// TIA Portal project "Moisture_meter" (V16)

(* hardware
DEVICE "S7-1200 station_1"  S7-1200 Station
   slot 0: "Rack_0"  S7-1200 Rack  Rack  V1.0
   slot 1: "PLC_1"  CPU 1215C DC/DC/DC  6ES7 215-1AG40-0XB0  V4.4
*)

// ===== PLC "PLC_1"  CPU 1215C DC/DC/DC =====

VAR_GLOBAL   // PLC tag table "Default tag table"
   "SW1Up" AT %I0.0 : Bool;   // Концевик-1 (верх)
   "SW2Up" AT %I0.1 : Bool;   // Концевик-2 (верх)
   "SW1Down" AT %I0.2 : Bool;   // Концевик-1 (Низ)
   "SW2Down" AT %I0.3 : Bool;   // Концевик-2 (Низ)
   "modeUp" AT %I0.4 : Bool;   // Режим (верх). Авто - True
   "modeDown" AT %I0.5 : Bool;   // Режим (Низ). Авто - True
   "EmergStop" AT %I0.6 : Bool;   // Аварийный стоп
   "readyDriveUp" AT %I0.7 : Bool;   // верхний драйвер ШД - Готов
   "alarmDriveUp" AT %I1.0 : Bool;   // верхний драйвер ШД - Авария
   "readyDriveDown" AT %I1.1 : Bool;   // Нижний драйвер ШД - Готов
   "alarmDriveDown" AT %I1.2 : Bool;   // Нижний драйвер ШД - Авария
   "Axis_1_Pulse" AT %Q0.0 : Bool;   // Импульсный выход для верхнего ШД
   "Axis_1_Direction" AT %Q0.1 : Bool;   // Направление вращения для верхнего ШД
   "Axis_2_Direction" AT %Q0.4 : Bool;   // Направление вращения для Нижнего ШД
   "Axis_2_Pulse" AT %Q0.3 : Bool;   // Импульсный выход для Нижнего ШД
   "disDriveUp" AT %Q0.2 : Bool;   // дективация драйвера шагового двигателя (верх)
   "disDriveDown" AT %Q0.5 : Bool;   // дективация драйвера шагового двигателя (Низ)
   "enAir" AT %Q0.6 : Bool;   // Подача воздуха
   "Tag_1" AT %M0.0 : Bool;
   "Tag_2" AT %M0.1 : Bool;
   "Tag_3" AT %M0.2 : Bool;
   "Tag_4" AT %M0.3 : Bool;
   "Tag_5" AT %M1.0 : Bool;
   "Tag_6" AT %M1.1 : Bool;
   "Tag_7" AT %M1.2 : Bool;
   "Axis_1_DriveEnable" AT %M6.0 : Bool;   // Активация верхнего драйвера ШД
   "Axis_2_DriveEnable" AT %M6.1 : Bool;   // Активация Нижнего драйвера ШД
   "Clock_Byte" AT %MB0 : Byte;
   "Clock_10Hz" AT %M0.0 : Bool;
   "Clock_5Hz" AT %M0.1 : Bool;
   "Clock_2.5Hz" AT %M0.2 : Bool;
   "Clock_2Hz" AT %M0.3 : Bool;
   "Clock_1.25Hz" AT %M0.4 : Bool;
   "Clock_1Hz" AT %M0.5 : Bool;
   "Clock_0.625Hz" AT %M0.6 : Bool;
   "Clock_0.5Hz" AT %M0.7 : Bool;
   "System_Byte" AT %MB1 : Byte;
   "FirstScan" AT %M1.0 : Bool;
   "DiagStatusUpdate" AT %M1.1 : Bool;
   "AlwaysTRUE" AT %M1.2 : Bool;
   "AlwaysFALSE" AT %M1.3 : Bool;
   "System_Byte(1)" AT %MB1 : Byte;
   "emergStopOut" AT %M7.0 : Bool;   // Сигнал Аварийный стоп без обработки
   "emergStopDelay" AT %M7.1 : Bool;   // Сигнал Аварийный стоп, задержка после снятия
   "emergStopPRG" AT %M7.2 : Bool;   // Сигнал Аварийный стоп для останова программных блоков
   "Tag_8" AT %M10.0 : Bool;
   "Tag_9" AT %M11.0 : Bool;
   "Tag_10" AT %M11.1 : Bool;
   "Tag_11" AT %M11.2 : Bool;
   "Tag_12" AT %M11.3 : Bool;
END_VAR

DATA_BLOCK "WRITE"   // DB5
{ S7_Optimized_Access := 'FALSE' }
VERSION : 0.1
   VAR
      airBlower : Bool := false;   // обдув кожуха и обектива
      upper : Struct
         jogForward : Bool := false;   // ручное движение вперед
         jogBackward : Bool := false;   // ручное движение назад
         width : DInt := 2050;   // ширина сканирования (100~2400mm)
         delay : DInt := 100;   // Задержка перед сменой направления
         speed : DInt := 50;   // Скорость движения (1~100%)
         speedJog : DInt := 50;   // Скорость движ. в ручном режиме
         speedInitia : DInt := 50;   // Скорость инициализации
         pulsesPerMeter : DInt := 170778;   // Импульсов на 1 метр
         offsetCenter : DInt := 0;   // смещение зоны сканирования относительно центра
      END_STRUCT;
      lower : Struct
         jogForward : Bool := false;   // ручное движение вперед
         jogBackward : Bool := false;   // ручное движение назад
         width : DInt := 2050;   // ширина сканирования (100~2400mm)
         delay : DInt := 100;   // Задержка перед сменой направления
         speed : DInt := 50;   // Скорость движения (1~100%)
         speedJog : DInt := 50;   // Скорость движ. в ручном режиме
         speedInitia : DInt := 50;   // Скорость инициализации
         pulsesPerMeter : DInt := 170778;   // Импульсов на 1 метр
         offsetCenter : DInt := 0;   // смещение зоны сканирования относительно центра
      END_STRUCT;
   END_VAR
BEGIN
END_DATA_BLOCK

DATA_BLOCK "Write_buffer"   // DB10
{ S7_Optimized_Access := 'FALSE' }
VERSION : 0.1
   VAR
      airBlower : Bool := false;   // обдув кожуха и обектива
      upper : Struct
         jogForward : Bool := false;   // ручное движение вперед
         jogBackward : Bool := false;   // ручное движение назад
         width : DInt := 2050;   // ширина сканирования (100~2400mm)
         delay : DInt := 100;   // Задержка перед сменой направления
         speed : DInt := 50;   // Скорость движения (1~100%)
         speedJog : DInt := 10;   // Скорость движ. в ручном режиме
         speedInitia : DInt := 5;   // Скорость инициализации
         pulsesPerMeter : DInt := 170778;   // Импульсов на 1 метр
         offsetCenter : DInt := 0;   // смещение зоны сканирования относительно центра
      END_STRUCT;
      lower : Struct
         jogForward : Bool := false;   // ручное движение вперед
         jogBackward : Bool := false;   // ручное движение назад
         width : DInt := 2050;   // ширина сканирования (100~2400mm)
         delay : DInt := 100;   // Задержка перед сменой направления
         speed : DInt := 50;   // Скорость движения (1~100%)
         speedJog : DInt := 10;   // Скорость движ. в ручном режиме
         speedInitia : DInt := 5;   // Скорость инициализации
         pulsesPerMeter : DInt := 170778;   // Импульсов на 1 метр
         offsetCenter : DInt := 0;   // смещение зоны сканирования относительно центра
      END_STRUCT;
   END_VAR
BEGIN
END_DATA_BLOCK

DATA_BLOCK "Edit_Input"   // DB11
{ S7_Optimized_Access := 'TRUE' }
VERSION : 0.1
   VAR
      SW1UpperEdit : USInt;   // 0 - выкл, 1 - False, 2 - True Концевик верх - 1
      SW2UpperEdit : USInt := 0;   // 0 - выкл, 1 - False, 2 - True Концевик верх - 2
      SW1lowerEdit : USInt := 0;   // 0 - выкл, 1 - False, 2 - True Концевик низ - 1
      SW2lowerEdit : USInt := 0;   // 0 - выкл, 1 - False, 2 - True Концевик низ - 2
      autoUpperEdit : USInt := 0;   // 0 - выкл, 1 - False, 2 - True Режим авто верх (вкл)
      autoLowerEdit : USInt := 0;   // 0 - выкл, 1 - False, 2 - True Режим авто Низ (вкл)
      emergencyStopEdit : USInt := 0;   // 0 - выкл, 1 - False, 2 - True Аварийный стоп
      readyUpperEdit : USInt := 0;   // 0 - выкл, 1 - False, 2 - True Привод верх - готов
      alarmUpperEdit : USInt := 0;   // 0 - выкл, 1 - False, 2 - True Привод верх - авария
      readyLowerEdit : USInt := 0;   // 0 - выкл, 1 - False, 2 - True Привод Низ - готов
      alarmlowerEdit : USInt := 0;   // 0 - выкл, 1 - False, 2 - True Привод Низ - авария
   END_VAR
BEGIN
END_DATA_BLOCK

DATA_BLOCK "READ"   // DB13
{ S7_Optimized_Access := 'FALSE' }
VERSION : 0.1
   VAR
      upper : Struct
         autoEn : Bool;   // задано авто перемещение
         status : USInt;   // 0: ожидание, 1: инициализация, 2: работа, 2:авария
         distanceL1 : DInt := 0;   // расстояние от нулевой позиции до начала обЪекта измерения, мм
         distanceL2 : DInt := 0;   // ширина обЪекта измерения, мм
         speed : DInt;   // скорость перемещения верхнего, %
         currDistance : DInt;   // положение влагомера на обЪекте измерения, мм
         currMoisture : Real;   // Текущая влажность
         arrayMoisture : Array[0..99] of Real;   // Массив влажности
      END_STRUCT;
      lower : Struct
         autoEn : Bool;   // задано авто перемещение
         status : USInt;   // 0: ожидание, 1: инициализация, 2: работа, 2:авария
         distanceL1 : DInt := 0;   // расстояние от нулевой позиции до начала обЪекта измерения, мм
         distanceL2 : DInt := 0;   // ширина обЪекта измерения, мм
         speed : DInt;   // скорость перемещения верхнего, %
         currDistance : DInt;   // положение влагомера на обЪекте измерения, мм
         currMoisture : Real;   // Текущая влажность
         arrayMoisture : Array[0..99] of Real;   // Массив влажности
      END_STRUCT;
      copyDbWrite : Struct
         airBlower : Bool := false;   // обдув кожуха и обектива
         upper : Struct
            jogForward : Bool := false;   // Премещение вперед (верх влагомер)
            jogBackward : Bool := false;   // Премещение Назад (верх влагомер)
            width : DInt := 2050;   // Длина пути рабоч. зоны (верхнего)
            delay : DInt := 100;   // Задержка перед сменой направления (верх)
            speed : DInt := 50;   // Скорость верхенего (%) от HMI
            speedJog : DInt := 10;   // Скорость движ. в ручном режиме верх
            speedInitia : DInt := 5;   // Скорость движ. при инициализации верх
            pulsesPerMeter : DInt := 170778;   // Импульсов на 1 метр от HMI (верхнего)
            offsetCenter : DInt := 0;   // коррекция длины L1 (верх)
         END_STRUCT;
         lower : Struct
            jogForward : Bool := false;   // Премещение вперед (низ влагомер)
            jogBackward : Bool := false;   // Премещение Назад (низ влагомер)
            width : DInt := 2050;   // Длина пути рабоч. зоны (нижнего)
            delay : DInt := 100;   // Задержка перед сменой направления (низ)
            speed : DInt := 50;   // Скорость нижнего (%) от HMI
            speedJog : DInt := 10;   // Скорость движ. в ручном режиме низ
            speedInitia : DInt := 5;   // Скорость движ. при инициализации низ
            pulsesPerMeter : DInt := 170778;   // Импульсов на 1 метр от HMI (нижнего)
            offsetCenter : DInt := 0;   // коррекция длины L1 (низ)
         END_STRUCT;
      END_STRUCT;
   END_VAR
BEGIN
END_DATA_BLOCK

DATA_BLOCK "main_DB"   // DB63
{ S7_Optimized_Access := 'FALSE' }
VERSION : 0.1
   VAR
      SW1Up : Bool;   // Концевик верх - 1
      SW2Up : Bool;   // Концевик верх - 2
      SW1Down : Bool;   // Концевик низ - 1
      SW2Down : Bool;   // Концевик низ - 2
      autoUp : Bool;   // Режим авто активен (верх). Активация авто перемещения.
      autoDown : Bool;   // Режим авто активен (Низ). Активация авто перемещения.
      readyDriveUp : Bool;   // Привод верх - готов
      alarmDriveUp : Bool;   // Привод верх - авария
      readyDriveDown : Bool;   // Привод Низ - готов
      alarmDriveDown : Bool;   // Привод Низ - авария
      modeInitiaUp : Bool;   // Статус - идет инициализация (верх)
      modeInitiaDown : Bool;   // Статус - идет инициализация (Низ)
      modeRunUp : Bool;   // Статус - активно авто перемещение (верх)
      modeRunDown : Bool;   // Статус - активно авто перемещение (Низ)
      directionUp : Bool;   // Направление движения. True - обратно (верх)
      directionDown : Bool;   // Направление движения. True - обратно (Низ)
      initializingUp : Bool;   // Флаг - инициализация (верх)
      initializingDown : Bool;   // Флаг - инициализация (Низ)
      initialOKUP : Bool;   // Инициализация завершена (без задержки) верх
      initialOKDown : Bool;   // Инициализация завершена (без задержки) Низ
      initialOKdelayUp : Bool;   // Инициализация завершена (с запазданием) верх
      initialOKdelayDown : Bool;   // Инициализация завершена (с запазданием) Низ
      "^ChangeL1Up" : Bool;   // Импульс если изменилось число L1 (верх)
      "^ChangeL2Up" : Bool;   // Импульс если изменилось число L2 (верх)
      "^ChangeL1Down" : Bool;   // Импульс если изменилось число L1 (Низ)
      "^ChangeL2Down" : Bool;   // Импульс если изменилось число L2 (Низ)
      disConnMoistUp : Bool;
      disConnMoistDown : Bool;
      modes : USInt;   // Код режимов для верха и низа (авто/руч)
      allStatus : USInt;   // Код общего состояния программы. 1 - экстренный стоп
      statusUpHMI : USInt;   // Код состояния программы верх 0 - ожидание, 1- сработал концевик, 2 - инициализация, 3 - работа, 4 - авария привода
      statusDownHMI : USInt;   // Код состояния программы Низ 0 - ожидание, 1- сработал концевик, 2 - инициализация, 3 - работа, 4 - авария привода
      speedJogMoveUp : DInt;   // Скорость (имп/сек). Принимает значение скорости при инициализации или ручного режима
      speedJogMoveDown : DInt;   // Скорость (имп/сек). Принимает значение скорости при инициализации или ручного режима
      pulsesPerMMUp : DInt;   // Вычисленное кол-во импульсов на 1мм пути (верх)
      pulsesPerMMDown : DInt;   // Вычисленное кол-во импульсов на 1мм пути (Низ)
      setPulsesUp : DInt;   // Текущая уставка длины L (верх)
      setPulsesDown : DInt;   // Текущая уставка длины L (Низ)
      actualPulsesUp : DInt;   // Текущая уставка длины L с инверсией знака для обратного движения (верх)
      actualPulsesDown : DInt;   // Текущая уставка длины L с инверсией знака для обратного движения (НИз)
      speedPulsesUp : DInt;   // Скорость перемещения в режиме авто (имп/сек) верх
      speedPulsesDown : DInt;   // Скорость перемещения в режиме авто (имп/сек) Низ
      speedPulsesIniUp : DInt;   // Скорость перемещения при инициализации (имп/сек) верх
      speedPulsesIniDown : DInt;   // Скорость перемещения при инициализации (имп/сек) Низ
      speedPulsesJogUp : DInt;   // Скорость перемещения в ручном режиме (имп/сек) верх
      speedPulsesJogDown : DInt;   // Скорость перемещения в ручном режиме (имп/сек) Низ
   END_VAR
BEGIN
END_DATA_BLOCK

// folder: FB_blocks

DATA_BLOCK "MBTCP2_DB"   // DB2
{ S7_Optimized_Access := 'TRUE' }
VERSION : 0.1
// stored: InstanceOfName MBTCP2
"MBTCP2"
BEGIN
END_DATA_BLOCK

DATA_BLOCK "MBTCP_1_DB"   // DB3
{ S7_Optimized_Access := 'TRUE' }
VERSION : 0.1
// stored: InstanceOfName MBTCP_1
"MBTCP_1"
BEGIN
END_DATA_BLOCK

DATA_BLOCK "Moisture_up_DB"   // DB7
{ S7_Optimized_Access := 'TRUE' }
VERSION : 0.1
// stored: InstanceOfName Moisture_array
"Moisture_array"
BEGIN
END_DATA_BLOCK

DATA_BLOCK "Moisture_down_DB"   // DB8
{ S7_Optimized_Access := 'TRUE' }
VERSION : 0.1
// stored: InstanceOfName Moisture_array
"Moisture_array"
BEGIN
END_DATA_BLOCK

// folder: Socket_Send

DATA_BLOCK "Send_Connect"   // DB17
{ S7_Optimized_Access := 'TRUE' }
AUTHOR : SIMATIC
FAMILY : MC7Plus
NAME : TC_IP_v4
VERSION : 1.0
// stored: InstanceOfName TCON_IP_v4
"TCON_IP_v4"
BEGIN
   ID := 4;
   InterfaceId := 64;
   LocalPort := 2000;
END_DATA_BLOCK

DATA_BLOCK "Sock_RD_DB"   // DB19
{ S7_Optimized_Access := 'TRUE' }
VERSION : 0.1
// stored: InstanceOfName Sock_RD
"Sock_RD"
BEGIN
END_DATA_BLOCK

// folder: Socket_Write

DATA_BLOCK "Sock_WR_db"   // DB9
{ S7_Optimized_Access := 'TRUE' }
VERSION : 0.1
// stored: InstanceOfName Sock_WR
"Sock_WR"
BEGIN
END_DATA_BLOCK

DATA_BLOCK "WriteBuffer"   // DB16
{ S7_Optimized_Access := 'FALSE' }
VERSION : 0.1
   VAR
      resetErrorTrigg : Bool;   // Сброс аварии
      coolAirEn : Bool;
      setLasersManual : Struct   // Для ручного режима
         upBlueLasers123 : Bool := false;
         upGreenLasers123 : Bool := false;
         upBlueLasers456 : Bool := false;
         upGreenLasers456 : Bool := false;
         upBlueLasers789 : Bool := false;
         downGreenLasers123 : Bool := false;
         downBlueLasers123 : Bool := false;
         downGreenLasers465 : Bool := false;
         downBlueLasers456 : Bool := false;
         downGreenLasers789 : Bool := false;
      END_STRUCT;
      simulate : Struct   // Симуляция каналов. (для АО применимо из setPowerLasers)
         DI : Struct
            DI0 : USInt := 16#0;
            DI1 : USInt := 16#0;
            DI2 : USInt := 16#0;
            DI3 : USInt := 16#0;
            DI4 : USInt := 16#0;
            DI5 : USInt := 16#0;
            DI6 : USInt := 16#0;
            DI7 : USInt := 16#0;
            DI8 : USInt := 16#0;
            DI9 : USInt := 16#0;
            DI10 : USInt := 16#0;
            DI11 : USInt := 16#0;
            DI12 : USInt := 16#0;
            DI13 : USInt := 16#0;
            DI14 : USInt := 16#0;
            DI15 : USInt := 16#0;
         END_STRUCT;
         "DO" : Struct
            DO0 : USInt := 0;
            DO1 : USInt := 0;
            DO2 : USInt := 0;
            DO3 : USInt := 0;
            DO4 : USInt := 0;
            DO5 : USInt := 0;
            DO6 : USInt := 0;
            DO7 : USInt := 0;
            DO8 : USInt := 0;
            DO9 : USInt := 0;
            DO10 : USInt := 0;
            DO11 : USInt := 0;
            DO12 : USInt := 0;
            DO13 : USInt := 0;
            DO14 : USInt := 0;
            DO15 : USInt := 0;
            DO16 : USInt := 0;
            DO17 : USInt := 0;
            DO18 : USInt := 0;
            DO19 : USInt := 0;
            DO20 : USInt := 0;
            DO21 : USInt := 0;
            DO22 : USInt := 0;
            DO23 : USInt := 0;
            DO24 : USInt := 0;
            DO25 : USInt := 0;
            DO26 : USInt := 0;
            DO27 : USInt := 0;
            DO28 : USInt := 0;
            DO29 : USInt := 0;
            DO30 : USInt := 0;
            DO31 : USInt := 0;
         END_STRUCT;
         AI : Struct   // 0.0 -- симуляция отключена; от 0.0 до 0.001 -- запись 0.0; выше 0.001 -- запись любого числа.
            upTempLaser1 : Real := 0.0;
            upTempLaser2 : Real := 0.0;
            upTempCam1 : Real := 0.0;
            upTempCam2 : Real := 0.0;
            downTempLaser1 : Real := 0.0;
            downTempLaser2 : Real := 0.0;
            downTempCam1 : Real := 0.0;
            downTempCam2 : Real := 0.0;
            airTemperatur : Real := 0.0;
            reserv : Real := 0.0;
         END_STRUCT;
      END_STRUCT;
      setTemperatures : Struct   // Уставки температур
         faultUpLaser : Real := 0.0;
         faultUpCam : Real := 0.0;
         faultDownLaser : Real := 0.0;
         faultDownCam : Real := 0.0;
         warnAir : Real := 0.0;
         warnUpLaser : Real := 0.0;
         warnUpCam : Real := 0.0;
         warnDownLaser : Real := 0.0;
         warnDownCam : Real := 0.0;
         reserv0 : Real := 0.0;
      END_STRUCT;
      cleanTime : Struct   // Периодичность продувки
         tOnS : Real := 0.0;
         tOffMin : Real := 0.0;
      END_STRUCT;
      setPowerLasers : Struct   // Мощность лазеров (0 -- 100%)
         writeAll : Real := 0.0;
         upBlue1 : Real := 0.0;   // AO0.0
         upBlue2 : Real := 0.0;   // AO0.1
         upBlue3 : Real := 0.0;   // AO0.2
         upGreen1 : Real := 0.0;   // AO0.3
         upGreen2 : Real := 0.0;   // AO0.4
         upGreen3 : Real := 0.0;   // AO0.5
         upBlue4 : Real := 0.0;   // AO0.6
         upBlue5 : Real := 0.0;   // AO0.7
         upBlue6 : Real := 0.0;   // AO1.0
         upGreen4 : Real := 0.0;   // AO1.1
         upGreen5 : Real := 0.0;   // AO1.2
         upGreen6 : Real := 0.0;   // AO1.3
         upBlue7 : Real := 0.0;   // AO1.4
         upBlue8 : Real := 0.0;   // AO1.5
         upBlue9 : Real := 0.0;   // AO1.6
         downGreen1 : Real := 0.0;   // AO2.0
         downGreen2 : Real := 0.0;   // AO2.1
         downGreen3 : Real := 0.0;   // AO2.2
         downBlue1 : Real := 0.0;   // AO2.3
         downBlue2 : Real := 0.0;   // AO2.4
         downBlue3 : Real := 0.0;   // AO2.5
         downGreen4 : Real := 0.0;   // AO2.6
         downGreen5 : Real := 0.0;   // AO2.7
         downGreen6 : Real := 0.0;   // AO3.0
         downBlue4 : Real := 0.0;   // AO3.1
         downBlue5 : Real := 0.0;   // AO3.2
         downBlue6 : Real := 0.0;   // AO3.3
         downGreen7 : Real := 0.0;   // AO3.4
         downGreen8 : Real := 0.0;   // AO3.5
         downGreen9 : Real := 0.0;   // AO3.6
      END_STRUCT;
   END_VAR
BEGIN
END_DATA_BLOCK

DATA_BLOCK "TRCV_Connect"   // DB20
{ S7_Optimized_Access := 'TRUE' }
AUTHOR : SIMATIC
FAMILY : MC7Plus
NAME : TC_IP_v4
VERSION : 1.0
// stored: InstanceOfName TCON_IP_v4
"TCON_IP_v4"
BEGIN
   ID := 3;
   InterfaceId := 64;
   LocalPort := 2001;
END_DATA_BLOCK

// folder: System blocks/Program resources

DATA_BLOCK "IEC_Timer_0_DB"   // DB14
{ S7_Optimized_Access := 'TRUE' }
AUTHOR : Simatic
FAMILY : IEC
NAME : IEC_TMR
VERSION : 1.0
// stored: InstanceOfName IEC_TIMER
"IEC_TIMER"
BEGIN
END_DATA_BLOCK

DATA_BLOCK "IEC_Timer_0_DB_1"   // DB15
{ S7_Optimized_Access := 'TRUE' }
AUTHOR : Simatic
FAMILY : IEC
NAME : IEC_TMR
VERSION : 1.0
// stored: InstanceOfName IEC_TIMER
"IEC_TIMER"
BEGIN
END_DATA_BLOCK

// folder: initializing

DATA_BLOCK "initializingUP_DB"   // DB12
{ S7_Optimized_Access := 'TRUE' }
VERSION : 0.1
// stored: InstanceOfName initializing
"initializing"
BEGIN
END_DATA_BLOCK

DATA_BLOCK "initializingDown_DB"   // DB60
{ S7_Optimized_Access := 'TRUE' }
VERSION : 0.1
// stored: InstanceOfName initializing
"initializing"
BEGIN
END_DATA_BLOCK

// folder: math

DATA_BLOCK "math_DB"   // DB25
{ S7_Optimized_Access := 'TRUE' }
VERSION : 0.1
// stored: InstanceOfName math
"math"
BEGIN
END_DATA_BLOCK

// folder: moving

DATA_BLOCK "movingUp_DB"   // DB26
{ S7_Optimized_Access := 'TRUE' }
VERSION : 0.1
// stored: InstanceOfName moving
"moving"
BEGIN
END_DATA_BLOCK

DATA_BLOCK "movingDown_DB"   // DB27
{ S7_Optimized_Access := 'TRUE' }
VERSION : 0.1
// stored: InstanceOfName moving
"moving"
BEGIN
END_DATA_BLOCK

// folder: status&Mode

DATA_BLOCK "statusMove_DB"   // DB4
{ S7_Optimized_Access := 'TRUE' }
VERSION : 0.1
// stored: InstanceOfName statusMove
"statusMove"
BEGIN
END_DATA_BLOCK

// folder: (top level)

DATA_BLOCK "AxisUpper"   // DB1, Motion_DB
{ S7_Optimized_Access := 'TRUE' }
AUTHOR : SIMATIC
FAMILY : BasicMC
NAME : TO_PosAx
VERSION : 7.0
// stored: InstanceOfName TO_PositioningAxis
"TO_PositioningAxis"
BEGIN
   // Axis.EnableOutput_AddressCU = %M6.0
   // Axis.DirectionOutputEnabledCU = TRUE
   // Axis.OnlinePtoModeCU = 16#0000_0002
   // Axis.SelectedChannel2EnumCU = %Q0.1
   // Axis.SelectedChannel1EnumCU = %Q0.0
   // Pulse.MinDeltaDeltaFrequencyCU = 0.004
   // Pulse.MaxDeltaDeltaFrequencyCU = 1.0E+10
   // Pulse.MinDeltaFrequencyCU = 0.005
   // Pulse.MaxDeltaFrequencyCU = 9.5E+9
   // Pulse.MinFrequencyCU = 1.0
   // Pulse.MaxFrequencyCU = 100000.0
   // Pulse.OutputSourceCU = 16#0000_0000
   // Axis.SelectPTO = 0
   // Axis.LengthUnit.LastDistance = -1
END_DATA_BLOCK

DATA_BLOCK "AxisLower"   // DB6, Motion_DB
{ S7_Optimized_Access := 'TRUE' }
AUTHOR : SIMATIC
FAMILY : BasicMC
NAME : TO_PosAx
VERSION : 7.0
// stored: InstanceOfName TO_PositioningAxis
"TO_PositioningAxis"
BEGIN
   // Axis.EnableOutput_AddressCU = %M6.1
   // Axis.LengthUnit.LastDistance = -1
   // Axis.DirectionOutputEnabledCU = TRUE
   // Axis.OnlinePtoModeCU = 16#0000_0002
   // Axis.SelectedChannel2EnumCU = %Q0.4
   // Axis.SelectedChannel1EnumCU = %Q0.3
   // Pulse.MinDeltaDeltaFrequencyCU = 0.004
   // Pulse.MaxDeltaDeltaFrequencyCU = 1.0E+10
   // Pulse.MinDeltaFrequencyCU = 0.005
   // Pulse.MaxDeltaFrequencyCU = 9.5E+9
   // Pulse.MinFrequencyCU = 1.0
   // Pulse.MaxFrequencyCU = 100000.0
   // Pulse.OutputSourceCU = 16#0000_0000
   // Axis.SelectPTO = 1
   // Axis.OnlinePtoIndexCU = 1
END_DATA_BLOCK

ORGANIZATION_BLOCK "Main"   // OB1, LAD, ProgramCycle
{ S7_Optimized_Access := 'TRUE' }
VERSION : 0.1
   VAR_INPUT
      Initial_Call : Bool;   // Initial call of this OB
      Remanence : Bool;   // =True, if remanent data are available
   END_VAR
BEGIN

REGION Network 1: Ручное изменение состояния дискретных входов контроллера
   // Значения хранятся в блоке Edit_Input [DB11]:    0 - выкл, 1 - False, 2 - True
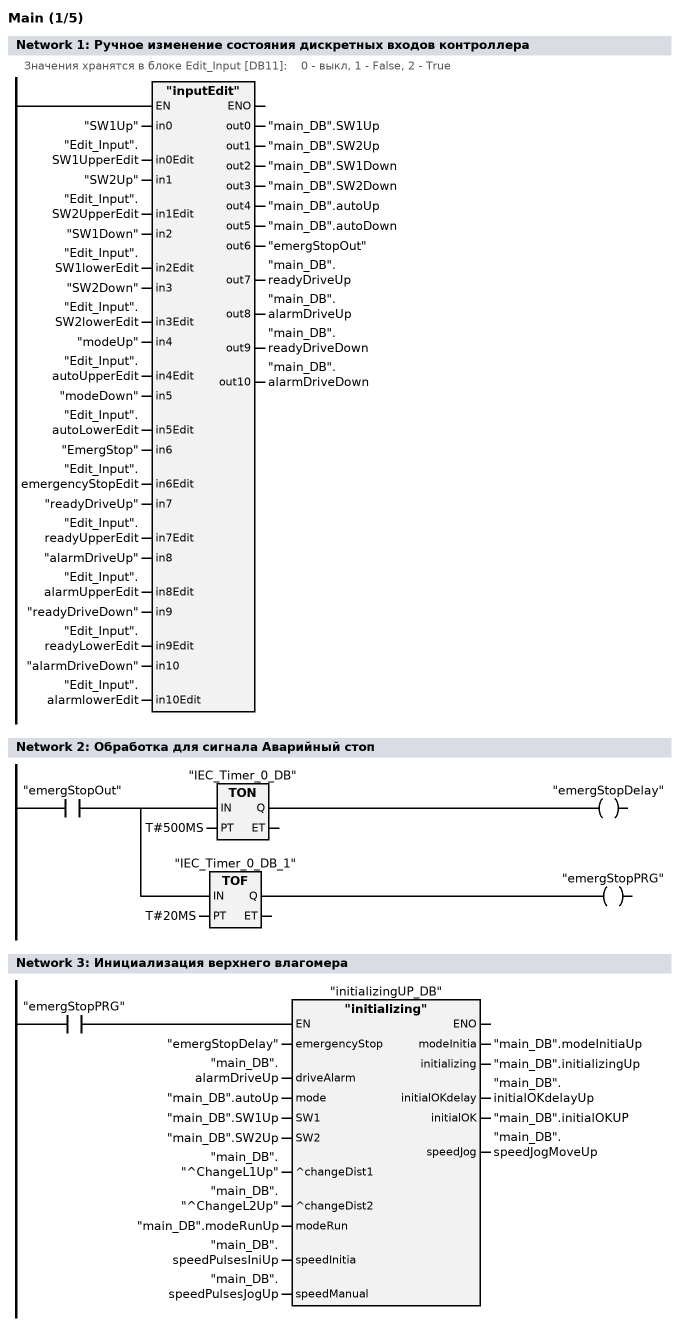
   RUNG wire#powerrail
      "inputEdit"(in0 := "SW1Up", in0Edit := "Edit_Input".SW1UpperEdit, in1 := "SW2Up", in1Edit := "Edit_Input".SW2UpperEdit, in2 := "SW1Down", in2Edit := "Edit_Input".SW1lowerEdit, in3 := "SW2Down", in3Edit := "Edit_Input".SW2lowerEdit, in4 := "modeUp", in4Edit := "Edit_Input".autoUpperEdit, in5 := "modeDown", in5Edit := "Edit_Input".autoLowerEdit, in6 := "EmergStop", in6Edit := "Edit_Input".emergencyStopEdit, in7 := "readyDriveUp", in7Edit := "Edit_Input".readyUpperEdit, in8 := "alarmDriveUp", in8Edit := "Edit_Input".alarmUpperEdit, in9 := "readyDriveDown", in9Edit := "Edit_Input".readyLowerEdit, in10 := "alarmDriveDown", in10Edit := "Edit_Input".alarmlowerEdit, out0 => "main_DB".SW1Up, out1 => "main_DB".SW2Up, out2 => "main_DB".SW1Down, out3 => "main_DB".SW2Down, out4 => "main_DB".autoUp, out5 => "main_DB".autoDown, out6 => "emergStopOut", out7 => "main_DB".readyDriveUp, out8 => "main_DB".alarmDriveUp, out9 => "main_DB".readyDriveDown, out10 => "main_DB".alarmDriveDown)
   END_RUNG
   // the same network as SCL:
   "inputEdit"(in0 := "SW1Up",
               in0Edit := "Edit_Input".SW1UpperEdit,
               in1 := "SW2Up",
               in1Edit := "Edit_Input".SW2UpperEdit,
               in2 := "SW1Down",
               in2Edit := "Edit_Input".SW1lowerEdit,
               in3 := "SW2Down",
               in3Edit := "Edit_Input".SW2lowerEdit,
               in4 := "modeUp",
               in4Edit := "Edit_Input".autoUpperEdit,
               in5 := "modeDown",
               in5Edit := "Edit_Input".autoLowerEdit,
               in6 := "EmergStop",
               in6Edit := "Edit_Input".emergencyStopEdit,
               in7 := "readyDriveUp",
               in7Edit := "Edit_Input".readyUpperEdit,
               in8 := "alarmDriveUp",
               in8Edit := "Edit_Input".alarmUpperEdit,
               in9 := "readyDriveDown",
               in9Edit := "Edit_Input".readyLowerEdit,
               in10 := "alarmDriveDown",
               in10Edit := "Edit_Input".alarmlowerEdit,
               out0 => "main_DB".SW1Up,
               out1 => "main_DB".SW2Up,
               out2 => "main_DB".SW1Down,
               out3 => "main_DB".SW2Down,
               out4 => "main_DB".autoUp,
               out5 => "main_DB".autoDown,
               out6 => "emergStopOut",
               out7 => "main_DB".readyDriveUp,
               out8 => "main_DB".alarmDriveUp,
               out9 => "main_DB".readyDriveDown,
               out10 => "main_DB".alarmDriveDown);
END_REGION

REGION Network 2: Обработка для сигнала Аварийный стоп
   "IEC_Timer_0_DB".TON(IN := "emergStopOut", PT := T#500MS);
   "emergStopDelay" := "IEC_Timer_0_DB".Q;
   "IEC_Timer_0_DB_1".TOF(IN := "emergStopOut", PT := T#20MS);
   "emergStopPRG" := "IEC_Timer_0_DB_1".Q;
END_REGION

REGION Network 3: Инициализация верхнего влагомера
   RUNG wire#powerrail
      Contact( "emergStopPRG" )
      "initializingUP_DB"(emergencyStop := "emergStopDelay", driveAlarm := "main_DB".alarmDriveUp, mode := "main_DB".autoUp, SW1 := "main_DB".SW1Up, SW2 := "main_DB".SW2Up, "^changeDist1" := "main_DB"."^ChangeL1Up", "^changeDist2" := "main_DB"."^ChangeL2Up", modeRun := "main_DB".modeRunUp, speedInitia := "main_DB".speedPulsesIniUp, speedManual := "main_DB".speedPulsesJogUp, modeInitia => "main_DB".modeInitiaUp, initializing => "main_DB".initializingUp, initialOKdelay => "main_DB".initialOKdelayUp, initialOK => "main_DB".initialOKUP, speedJog => "main_DB".speedJogMoveUp)
   END_RUNG
   // the same network as SCL:
   IF "emergStopPRG" THEN
       "initializingUP_DB"(emergencyStop := "emergStopDelay",   // "initializing"
                           driveAlarm := "main_DB".alarmDriveUp,
                           mode := "main_DB".autoUp,
                           SW1 := "main_DB".SW1Up,
                           SW2 := "main_DB".SW2Up,
                           "^changeDist1" := "main_DB"."^ChangeL1Up",
                           "^changeDist2" := "main_DB"."^ChangeL2Up",
                           modeRun := "main_DB".modeRunUp,
                           speedInitia := "main_DB".speedPulsesIniUp,
                           speedManual := "main_DB".speedPulsesJogUp,
                           modeInitia => "main_DB".modeInitiaUp,
                           initializing => "main_DB".initializingUp,
                           initialOKdelay => "main_DB".initialOKdelayUp,
                           initialOK => "main_DB".initialOKUP,
                           speedJog => "main_DB".speedJogMoveUp);
   END_IF;
END_REGION

REGION Network 4: Инициализация нижнего влагомера
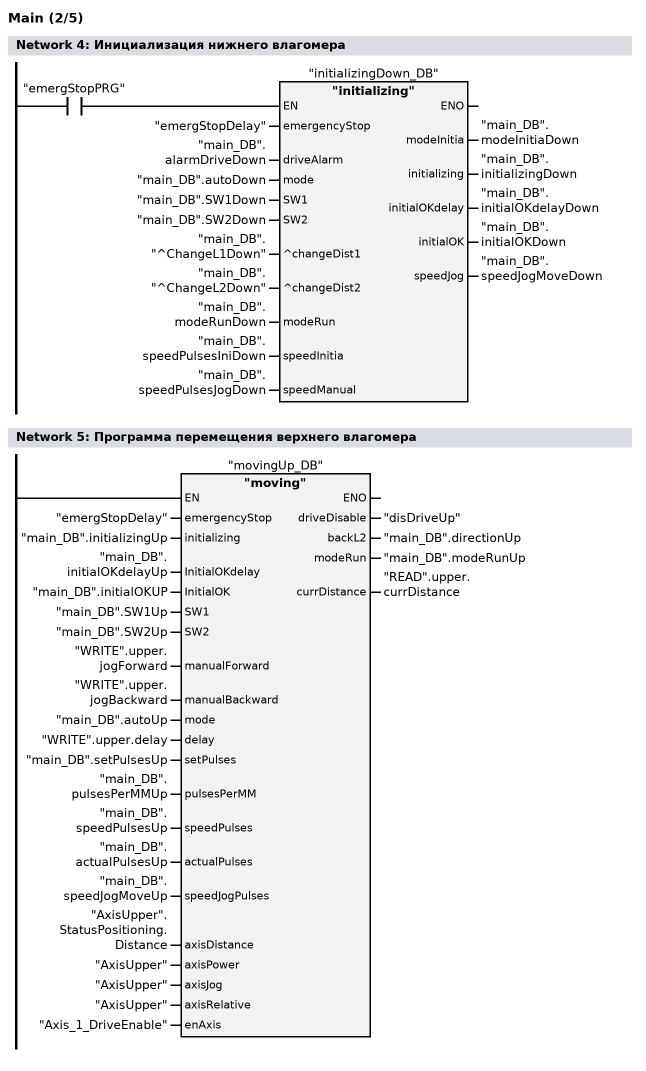
   RUNG wire#powerrail
      Contact( "emergStopPRG" )
      "initializingDown_DB"(emergencyStop := "emergStopDelay", driveAlarm := "main_DB".alarmDriveDown, mode := "main_DB".autoDown, SW1 := "main_DB".SW1Down, SW2 := "main_DB".SW2Down, "^changeDist1" := "main_DB"."^ChangeL1Down", "^changeDist2" := "main_DB"."^ChangeL2Down", modeRun := "main_DB".modeRunDown, speedInitia := "main_DB".speedPulsesIniDown, speedManual := "main_DB".speedPulsesJogDown, modeInitia => "main_DB".modeInitiaDown, initializing => "main_DB".initializingDown, initialOKdelay => "main_DB".initialOKdelayDown, initialOK => "main_DB".initialOKDown, speedJog => "main_DB".speedJogMoveDown)
   END_RUNG
   // the same network as SCL:
   IF "emergStopPRG" THEN
       "initializingDown_DB"(emergencyStop := "emergStopDelay",   // "initializing"
                             driveAlarm := "main_DB".alarmDriveDown,
                             mode := "main_DB".autoDown,
                             SW1 := "main_DB".SW1Down,
                             SW2 := "main_DB".SW2Down,
                             "^changeDist1" := "main_DB"."^ChangeL1Down",
                             "^changeDist2" := "main_DB"."^ChangeL2Down",
                             modeRun := "main_DB".modeRunDown,
                             speedInitia := "main_DB".speedPulsesIniDown,
                             speedManual := "main_DB".speedPulsesJogDown,
                             modeInitia => "main_DB".modeInitiaDown,
                             initializing => "main_DB".initializingDown,
                             initialOKdelay => "main_DB".initialOKdelayDown,
                             initialOK => "main_DB".initialOKDown,
                             speedJog => "main_DB".speedJogMoveDown);
   END_IF;
END_REGION

REGION Network 5: Программа перемещения верхнего влагомера
   RUNG wire#powerrail
      "movingUp_DB"(emergencyStop := "emergStopDelay", initializing := "main_DB".initializingUp, InitialOKdelay := "main_DB".initialOKdelayUp, InitialOK := "main_DB".initialOKUP, SW1 := "main_DB".SW1Up, SW2 := "main_DB".SW2Up, manualForward := "WRITE".upper.jogForward, manualBackward := "WRITE".upper.jogBackward, mode := "main_DB".autoUp, delay := "WRITE".upper.delay, setPulses := "main_DB".setPulsesUp, pulsesPerMM := "main_DB".pulsesPerMMUp, speedPulses := "main_DB".speedPulsesUp, actualPulses := "main_DB".actualPulsesUp, speedJogPulses := "main_DB".speedJogMoveUp, axisDistance := "AxisUpper".StatusPositioning.Distance, axisPower := "AxisUpper", axisJog := "AxisUpper", axisRelative := "AxisUpper", enAxis := "Axis_1_DriveEnable", driveDisable => "disDriveUp", backL2 => "main_DB".directionUp, modeRun => "main_DB".modeRunUp, currDistance => "READ".upper.currDistance)
   END_RUNG
   // the same network as SCL:
   "movingUp_DB"(emergencyStop := "emergStopDelay",   // "moving"
                 initializing := "main_DB".initializingUp,
                 InitialOKdelay := "main_DB".initialOKdelayUp,
                 InitialOK := "main_DB".initialOKUP,
                 SW1 := "main_DB".SW1Up,
                 SW2 := "main_DB".SW2Up,
                 manualForward := "WRITE".upper.jogForward,
                 manualBackward := "WRITE".upper.jogBackward,
                 mode := "main_DB".autoUp,
                 delay := "WRITE".upper.delay,
                 setPulses := "main_DB".setPulsesUp,
                 pulsesPerMM := "main_DB".pulsesPerMMUp,
                 speedPulses := "main_DB".speedPulsesUp,
                 actualPulses := "main_DB".actualPulsesUp,
                 speedJogPulses := "main_DB".speedJogMoveUp,
                 axisDistance := "AxisUpper".StatusPositioning.Distance,
                 axisPower := "AxisUpper",
                 axisJog := "AxisUpper",
                 axisRelative := "AxisUpper",
                 enAxis := "Axis_1_DriveEnable",
                 driveDisable => "disDriveUp",
                 backL2 => "main_DB".directionUp,
                 modeRun => "main_DB".modeRunUp,
                 currDistance => "READ".upper.currDistance);
END_REGION

REGION Network 6: Программа перемещения нижнего влагомера
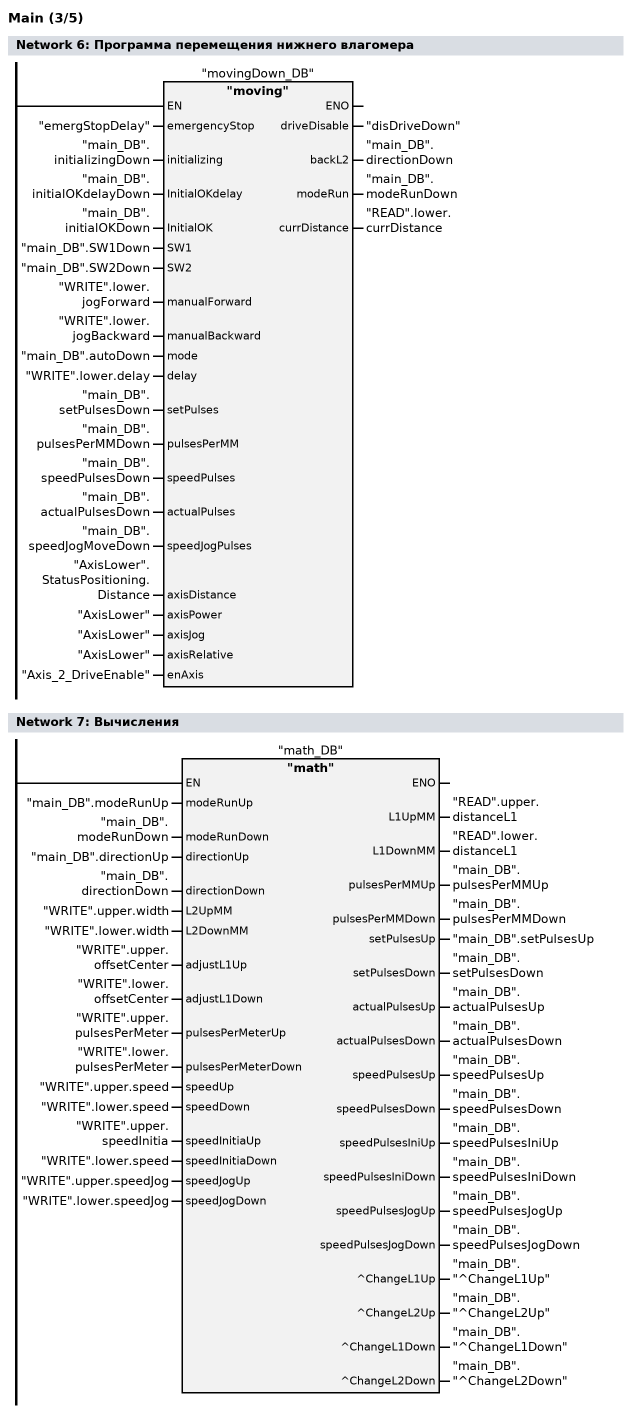
   RUNG wire#powerrail
      "movingDown_DB"(emergencyStop := "emergStopDelay", initializing := "main_DB".initializingDown, InitialOKdelay := "main_DB".initialOKdelayDown, InitialOK := "main_DB".initialOKDown, SW1 := "main_DB".SW1Down, SW2 := "main_DB".SW2Down, manualForward := "WRITE".lower.jogForward, manualBackward := "WRITE".lower.jogBackward, mode := "main_DB".autoDown, delay := "WRITE".lower.delay, setPulses := "main_DB".setPulsesDown, pulsesPerMM := "main_DB".pulsesPerMMDown, speedPulses := "main_DB".speedPulsesDown, actualPulses := "main_DB".actualPulsesDown, speedJogPulses := "main_DB".speedJogMoveDown, axisDistance := "AxisLower".StatusPositioning.Distance, axisPower := "AxisLower", axisJog := "AxisLower", axisRelative := "AxisLower", enAxis := "Axis_2_DriveEnable", driveDisable => "disDriveDown", backL2 => "main_DB".directionDown, modeRun => "main_DB".modeRunDown, currDistance => "READ".lower.currDistance)
   END_RUNG
   // the same network as SCL:
   "movingDown_DB"(emergencyStop := "emergStopDelay",   // "moving"
                   initializing := "main_DB".initializingDown,
                   InitialOKdelay := "main_DB".initialOKdelayDown,
                   InitialOK := "main_DB".initialOKDown,
                   SW1 := "main_DB".SW1Down,
                   SW2 := "main_DB".SW2Down,
                   manualForward := "WRITE".lower.jogForward,
                   manualBackward := "WRITE".lower.jogBackward,
                   mode := "main_DB".autoDown,
                   delay := "WRITE".lower.delay,
                   setPulses := "main_DB".setPulsesDown,
                   pulsesPerMM := "main_DB".pulsesPerMMDown,
                   speedPulses := "main_DB".speedPulsesDown,
                   actualPulses := "main_DB".actualPulsesDown,
                   speedJogPulses := "main_DB".speedJogMoveDown,
                   axisDistance := "AxisLower".StatusPositioning.Distance,
                   axisPower := "AxisLower",
                   axisJog := "AxisLower",
                   axisRelative := "AxisLower",
                   enAxis := "Axis_2_DriveEnable",
                   driveDisable => "disDriveDown",
                   backL2 => "main_DB".directionDown,
                   modeRun => "main_DB".modeRunDown,
                   currDistance => "READ".lower.currDistance);
END_REGION

REGION Network 7: Вычисления
   RUNG wire#powerrail
      "math_DB"(modeRunUp := "main_DB".modeRunUp, modeRunDown := "main_DB".modeRunDown, directionUp := "main_DB".directionUp, directionDown := "main_DB".directionDown, L2UpMM := "WRITE".upper.width, L2DownMM := "WRITE".lower.width, adjustL1Up := "WRITE".upper.offsetCenter, adjustL1Down := "WRITE".lower.offsetCenter, pulsesPerMeterUp := "WRITE".upper.pulsesPerMeter, pulsesPerMeterDown := "WRITE".lower.pulsesPerMeter, speedUp := "WRITE".upper.speed, speedDown := "WRITE".lower.speed, speedInitiaUp := "WRITE".upper.speedInitia, speedInitiaDown := "WRITE".lower.speed, speedJogUp := "WRITE".upper.speedJog, speedJogDown := "WRITE".lower.speedJog, L1UpMM => "READ".upper.distanceL1, L1DownMM => "READ".lower.distanceL1, pulsesPerMMUp => "main_DB".pulsesPerMMUp, pulsesPerMMDown => "main_DB".pulsesPerMMDown, setPulsesUp => "main_DB".setPulsesUp, setPulsesDown => "main_DB".setPulsesDown, actualPulsesUp => "main_DB".actualPulsesUp, actualPulsesDown => "main_DB".actualPulsesDown, speedPulsesUp => "main_DB".speedPulsesUp, speedPulsesDown => "main_DB".speedPulsesDown, speedPulsesIniUp => "main_DB".speedPulsesIniUp, speedPulsesIniDown => "main_DB".speedPulsesIniDown, speedPulsesJogUp => "main_DB".speedPulsesJogUp, speedPulsesJogDown => "main_DB".speedPulsesJogDown, "^ChangeL1Up" => "main_DB"."^ChangeL1Up", "^ChangeL2Up" => "main_DB"."^ChangeL2Up", "^ChangeL1Down" => "main_DB"."^ChangeL1Down", "^ChangeL2Down" => "main_DB"."^ChangeL2Down")
   END_RUNG
   // the same network as SCL:
   "math_DB"(modeRunUp := "main_DB".modeRunUp,   // "math"
             modeRunDown := "main_DB".modeRunDown,
             directionUp := "main_DB".directionUp,
             directionDown := "main_DB".directionDown,
             L2UpMM := "WRITE".upper.width,
             L2DownMM := "WRITE".lower.width,
             adjustL1Up := "WRITE".upper.offsetCenter,
             adjustL1Down := "WRITE".lower.offsetCenter,
             pulsesPerMeterUp := "WRITE".upper.pulsesPerMeter,
             pulsesPerMeterDown := "WRITE".lower.pulsesPerMeter,
             speedUp := "WRITE".upper.speed,
             speedDown := "WRITE".lower.speed,
             speedInitiaUp := "WRITE".upper.speedInitia,
             speedInitiaDown := "WRITE".lower.speed,
             speedJogUp := "WRITE".upper.speedJog,
             speedJogDown := "WRITE".lower.speedJog,
             L1UpMM => "READ".upper.distanceL1,
             L1DownMM => "READ".lower.distanceL1,
             pulsesPerMMUp => "main_DB".pulsesPerMMUp,
             pulsesPerMMDown => "main_DB".pulsesPerMMDown,
             setPulsesUp => "main_DB".setPulsesUp,
             setPulsesDown => "main_DB".setPulsesDown,
             actualPulsesUp => "main_DB".actualPulsesUp,
             actualPulsesDown => "main_DB".actualPulsesDown,
             speedPulsesUp => "main_DB".speedPulsesUp,
             speedPulsesDown => "main_DB".speedPulsesDown,
             speedPulsesIniUp => "main_DB".speedPulsesIniUp,
             speedPulsesIniDown => "main_DB".speedPulsesIniDown,
             speedPulsesJogUp => "main_DB".speedPulsesJogUp,
             speedPulsesJogDown => "main_DB".speedPulsesJogDown,
             "^ChangeL1Up" => "main_DB"."^ChangeL1Up",
             "^ChangeL2Up" => "main_DB"."^ChangeL2Up",
             "^ChangeL1Down" => "main_DB"."^ChangeL1Down",
             "^ChangeL2Down" => "main_DB"."^ChangeL2Down");
END_REGION

REGION Network 8: Статусы программ и передача между блоками данных
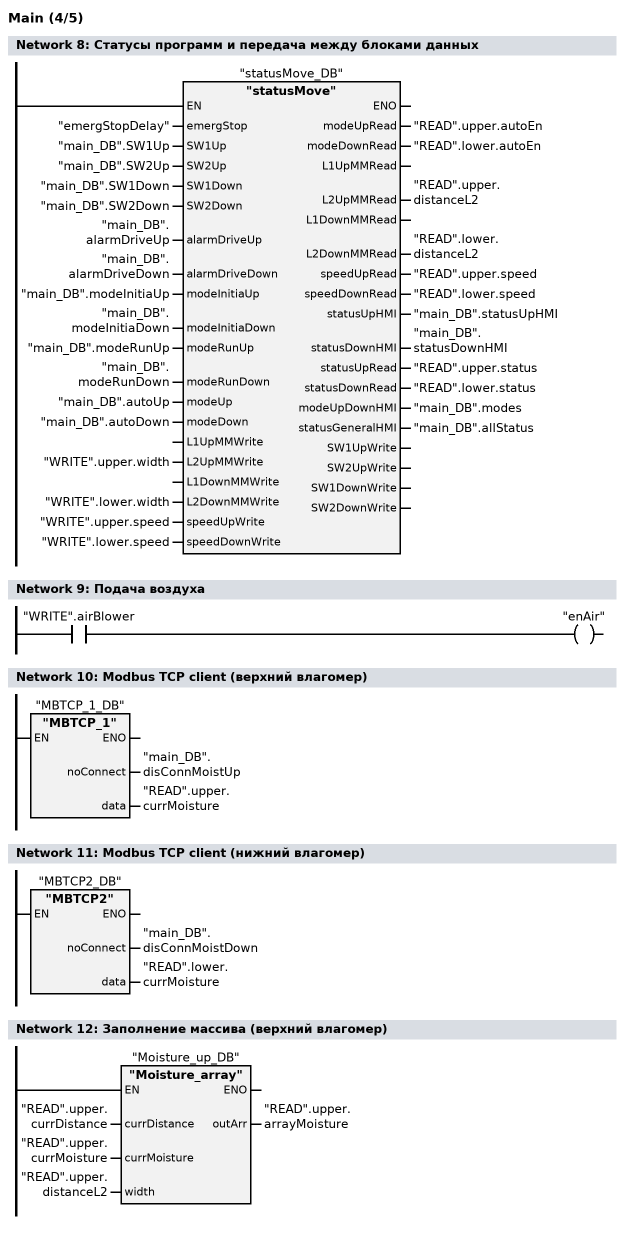
   RUNG wire#powerrail
      "statusMove_DB"(emergStop := "emergStopDelay", SW1Up := "main_DB".SW1Up, SW2Up := "main_DB".SW2Up, SW1Down := "main_DB".SW1Down, SW2Down := "main_DB".SW2Down, alarmDriveUp := "main_DB".alarmDriveUp, alarmDriveDown := "main_DB".alarmDriveDown, modeInitiaUp := "main_DB".modeInitiaUp, modeInitiaDown := "main_DB".modeInitiaDown, modeRunUp := "main_DB".modeRunUp, modeRunDown := "main_DB".modeRunDown, modeUp := "main_DB".autoUp, modeDown := "main_DB".autoDown, L1UpMMWrite :=, L2UpMMWrite := "WRITE".upper.width, L1DownMMWrite :=, L2DownMMWrite := "WRITE".lower.width, speedUpWrite := "WRITE".upper.speed, speedDownWrite := "WRITE".lower.speed, modeUpRead => "READ".upper.autoEn, modeDownRead => "READ".lower.autoEn, L1UpMMRead =>, L2UpMMRead => "READ".upper.distanceL2, L1DownMMRead =>, L2DownMMRead => "READ".lower.distanceL2, speedUpRead => "READ".upper.speed, speedDownRead => "READ".lower.speed, statusUpHMI => "main_DB".statusUpHMI, statusDownHMI => "main_DB".statusDownHMI, statusUpRead => "READ".upper.status, statusDownRead => "READ".lower.status, modeUpDownHMI => "main_DB".modes, statusGeneralHMI => "main_DB".allStatus, SW1UpWrite =>, SW2UpWrite =>, SW1DownWrite =>, SW2DownWrite =>)
   END_RUNG
   // the same network as SCL:
   "statusMove_DB"(emergStop := "emergStopDelay",   // "statusMove"
                   SW1Up := "main_DB".SW1Up,
                   SW2Up := "main_DB".SW2Up,
                   SW1Down := "main_DB".SW1Down,
                   SW2Down := "main_DB".SW2Down,
                   alarmDriveUp := "main_DB".alarmDriveUp,
                   alarmDriveDown := "main_DB".alarmDriveDown,
                   modeInitiaUp := "main_DB".modeInitiaUp,
                   modeInitiaDown := "main_DB".modeInitiaDown,
                   modeRunUp := "main_DB".modeRunUp,
                   modeRunDown := "main_DB".modeRunDown,
                   modeUp := "main_DB".autoUp,
                   modeDown := "main_DB".autoDown,
                   L2UpMMWrite := "WRITE".upper.width,
                   L2DownMMWrite := "WRITE".lower.width,
                   speedUpWrite := "WRITE".upper.speed,
                   speedDownWrite := "WRITE".lower.speed,
                   modeUpRead => "READ".upper.autoEn,
                   modeDownRead => "READ".lower.autoEn,
                   L2UpMMRead => "READ".upper.distanceL2,
                   L2DownMMRead => "READ".lower.distanceL2,
                   speedUpRead => "READ".upper.speed,
                   speedDownRead => "READ".lower.speed,
                   statusUpHMI => "main_DB".statusUpHMI,
                   statusDownHMI => "main_DB".statusDownHMI,
                   statusUpRead => "READ".upper.status,
                   statusDownRead => "READ".lower.status,
                   modeUpDownHMI => "main_DB".modes,
                   statusGeneralHMI => "main_DB".allStatus);
END_REGION

REGION Network 9: Подача воздуха
   RUNG wire#powerrail
      Contact( "WRITE".airBlower )
      Coil( "enAir" )
   END_RUNG
   // the same network as SCL:
   "enAir" := "WRITE".airBlower;
END_REGION

REGION Network 10: Modbus TCP client (верхний влагомер)
   RUNG wire#powerrail
      "MBTCP_1_DB"(noConnect => "main_DB".disConnMoistUp, data => "READ".upper.currMoisture)
   END_RUNG
   // the same network as SCL:
   "MBTCP_1_DB"(noConnect => "main_DB".disConnMoistUp, data => "READ".upper.currMoisture);   // "MBTCP_1"
END_REGION

REGION Network 11: Modbus TCP client (нижний влагомер)
   RUNG wire#powerrail
      "MBTCP2_DB"(noConnect => "main_DB".disConnMoistDown, data => "READ".lower.currMoisture)
   END_RUNG
   // the same network as SCL:
   "MBTCP2_DB"(noConnect => "main_DB".disConnMoistDown, data => "READ".lower.currMoisture);   // "MBTCP2"
END_REGION

REGION Network 12: Заполнение массива (верхний влагомер)
   RUNG wire#powerrail
      "Moisture_up_DB"(currDistance := "READ".upper.currDistance, currMoisture := "READ".upper.currMoisture, width := "READ".upper.distanceL2, outArr => "READ".upper.arrayMoisture)
   END_RUNG
   // the same network as SCL:
   "Moisture_up_DB"(currDistance := "READ".upper.currDistance,   // "Moisture_array"
                    currMoisture := "READ".upper.currMoisture,
                    width := "READ".upper.distanceL2,
                    outArr => "READ".upper.arrayMoisture);
END_REGION

REGION Network 13: Заполнение массива (нижний влагомер)
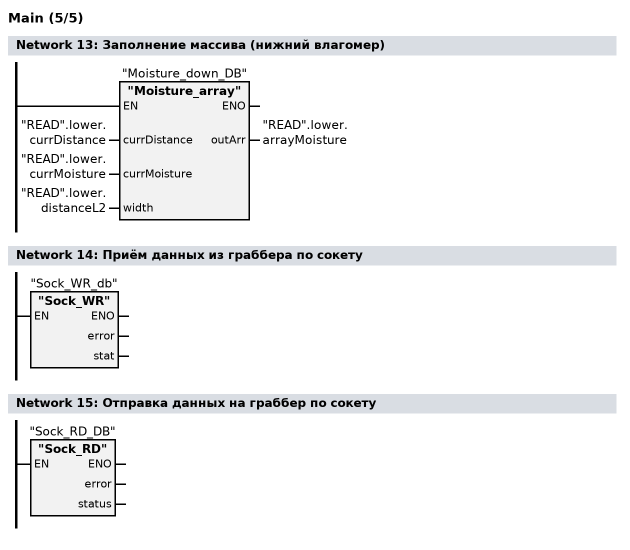
   RUNG wire#powerrail
      "Moisture_down_DB"(currDistance := "READ".lower.currDistance, currMoisture := "READ".lower.currMoisture, width := "READ".lower.distanceL2, outArr => "READ".lower.arrayMoisture)
   END_RUNG
   // the same network as SCL:
   "Moisture_down_DB"(currDistance := "READ".lower.currDistance,   // "Moisture_array"
                      currMoisture := "READ".lower.currMoisture,
                      width := "READ".lower.distanceL2,
                      outArr => "READ".lower.arrayMoisture);
END_REGION

REGION Network 14: Приём данных из граббера по сокету
   RUNG wire#powerrail
      "Sock_WR_db"(error =>, stat =>)
   END_RUNG
   // the same network as SCL:
   "Sock_WR_db"();   // "Sock_WR"
END_REGION

REGION Network 15: Отправка данных на граббер по сокету
   RUNG wire#powerrail
      "Sock_RD_DB"(error =>, status =>)
   END_RUNG
   // the same network as SCL:
   "Sock_RD_DB"();   // "Sock_RD"
END_REGION
END_ORGANIZATION_BLOCK

// folder: FB_blocks

FUNCTION_BLOCK "^Ch_Dint"   // FB1, SCL
{ S7_Optimized_Access := 'TRUE' }
VERSION : 0.1
   VAR_INPUT
      in : DInt;
   END_VAR
   VAR_OUTPUT
      "^out" : Bool;
   END_VAR
   VAR
      buff : DInt;
   END_VAR
BEGIN
   IF #in <> #buff THEN
       #"^out" := true;
   ELSE
       #"^out" := false;
   END_IF;
   #buff := #in;
END_FUNCTION_BLOCK

FUNCTION_BLOCK "Moisture_array"   // FB3, LAD
{ S7_Optimized_Access := 'TRUE' }
VERSION : 0.1
   VAR_INPUT
      currDistance : DInt;
      currMoisture : Real;
      width : DInt;
   END_VAR
   VAR_OUTPUT
      outArr : Array[0..99] of Real;
   END_VAR
   VAR
      buffArr : Array[0..99] of Real;
      writeOk : Bool;
      ds : Array[0..99] of Real;
      i : Int;
   END_VAR
   VAR_TEMP
      numArr : Int;
   END_VAR
BEGIN

REGION Network 1 (SCL)
   // Расчет элемента массива исходя из текущей дистанции и формата сырья
   // С лимитом, для защиты от некорректного числа
   #buffArr[LIMIT(MN := 0, IN := #currDistance * 99 / #width, MX := 99)] := #currMoisture;

   // Запись один цикл в крайних положениях
   IF (#currDistance = 0 OR #currDistance = #width) AND NOT #writeOk THEN
       #outArr := #buffArr;
       #writeOk := True;
   ELSIF #currDistance > 0 AND #currDistance < #width THEN
       #writeOk := False;
   END_IF;
END_REGION
END_FUNCTION_BLOCK

FUNCTION_BLOCK "CurrDistance"   // FB4, SCL
{ S7_Optimized_Access := 'TRUE' }
VERSION : 0.1
   VAR_INPUT
      En_1 : Bool;
      forward : Bool;
      backward : Bool;
      done : Bool;
      Distance : Real;
      ActualDistance : Real;
      PulsesPerMm : Real;
   END_VAR
   VAR_OUTPUT
      currDistanceMm : DInt;
   END_VAR
   VAR
      Sel0 : Real;
      Sel1 : Real;
      Sel2 : Real;
      Sel3 : Real;
      Sel4 : Real := 0.0;
      DoneDel : Bool;
      CalcDictance : Real;
      R_TRIG_Instance : R_TRIG;
      R_TRIG_Instance_1 : R_TRIG;
   END_VAR
   VAR_TEMP
      "^Forward" : Bool;
      "^Backward" : Bool;
      "Forward^" : Bool;
      "Backward^" : Bool;
   END_VAR
BEGIN
   #R_TRIG_Instance(CLK:=#forward,
                    Q=>#"^Forward"); // фронт сигнала forward
   #R_TRIG_Instance_1(CLK:=#backward,
                      Q=>#"^Backward");// фронт сигнала backward

   #CalcDictance := (#Distance - #ActualDistance); // Вычисляем пройденный путь

   REGION Триггер для числа CalcDictance. Set - #forward AND NOT #Done. Reset - #"^Forward" OR NOT #En_1)
       #Sel0 := SEL(G := #"^Forward" OR NOT #En_1, IN0 := #Sel1, IN1 := 0);
       #Sel1 := SEL(G := #forward AND NOT #DoneDel, IN0 := #Sel0, IN1 := #CalcDictance);
   END_REGION

   REGION Триггер для числа CalcDictance. Set -  #backward AND NOT #Done.   Reset - #"^Backward" OR #"^Forward".
       #Sel2 := SEL(G := #"^Backward" OR #"^Forward" OR NOT #En_1, IN0 := #Sel3, IN1 := 0);
       #Sel3 := SEL(G := #backward AND NOT #DoneDel, IN0 := #Sel2, IN1 := #CalcDictance);
   END_REGION

   #currDistanceMm := (#Sel0 - #Sel2) / #PulsesPerMm; // результат в переводе в мм (целое число)

   #DoneDel := #done; // DoneDel - (Done с запазданием на один цикл) 

   IF #ActualDistance = 0 THEN
       #CalcDictance := 0;
   END_IF; // на всякий случай обнуляем
END_FUNCTION_BLOCK

FUNCTION_BLOCK "MBTCP_1"   // FB9, SCL
{ S7_Optimized_Access := 'TRUE' }
VERSION : 0.1
   VAR_OUTPUT
      noConnect : Bool := false;
      data : Real := 0.0;
   END_VAR
   VAR
      Srv1Disconect : Bool := false;
      request : Bool;
      count : Int;
      modbus0 : MB_CLIENT;
      Server1_connect : TCON_IP_v4;
      TOF0 : TOF_TIME;
   END_VAR
   // Server1_connect.InterfaceId := 64;
   // Server1_connect.ID := 1;
   // Server1_connect.ConnectionType := 11;
   // Server1_connect.ActiveEstablished := true;
   // Server1_connect.RemoteAddress.ADDR[1] := 192;
   // Server1_connect.RemoteAddress.ADDR[2] := 168;
   // Server1_connect.RemoteAddress.ADDR[3] := 113;
   // Server1_connect.RemoteAddress.ADDR[4] := 53;
   // Server1_connect.RemotePort := 8000;
   // Server1_connect.LocalPort := 0;
BEGIN

   #request := NOT #request;

   #modbus0(REQ := #request,
                DISCONNECT := #Srv1Disconect,
                MB_MODE := 0,
                MB_DATA_ADDR := 40388,
                MB_DATA_LEN := 2,
                MB_DATA_PTR := #data,
                CONNECT := #Server1_connect);


   #TOF0(IN:=#modbus0.ERROR OR (#modbus0.STATUS = 16#7002),
                         PT:=T#700MS,
                         Q=>#noConnect);
END_FUNCTION_BLOCK

FUNCTION_BLOCK "MBTCP2"   // FB10, SCL
{ S7_Optimized_Access := 'TRUE' }
VERSION : 0.1
   VAR_OUTPUT
      noConnect : Bool;
      data : Real;
   END_VAR
   VAR
      Server2_connect : TCON_IP_v4;
      TOF0 : TOF_TIME;
      Srv1Disconect : Bool := false;
      request : Bool;
      Srv1Status : Word;
      modbus0 : MB_CLIENT;
   END_VAR
   // Server2_connect.InterfaceId := 64;
   // Server2_connect.ID := 2;
   // Server2_connect.ConnectionType := 11;
   // Server2_connect.ActiveEstablished := true;
   // Server2_connect.RemoteAddress.ADDR[1] := 192;
   // Server2_connect.RemoteAddress.ADDR[2] := 168;
   // Server2_connect.RemoteAddress.ADDR[3] := 113;
   // Server2_connect.RemoteAddress.ADDR[4] := 54;
   // Server2_connect.RemotePort := 8000;
   // Server2_connect.LocalPort := 0;
BEGIN

   #request := NOT #request;

   #modbus0(REQ := #request,
                DISCONNECT := #Srv1Disconect,
                MB_MODE := 0,
                MB_DATA_ADDR := 40388,
                MB_DATA_LEN := 2,
                MB_DATA_PTR := #data,
                CONNECT := #Server2_connect);


   #TOF0(IN:=#modbus0.ERROR OR (#modbus0.STATUS = 16#7002),
         PT:=T#700MS,
         Q=>#noConnect);
END_FUNCTION_BLOCK

// folder: Socket_Send

FUNCTION_BLOCK "Sock_RD"   // FB12, LAD
{ S7_Optimized_Access := 'TRUE' }
VERSION : 0.1
   VAR_OUTPUT
      error : Bool;
      status : Word;
   END_VAR
   VAR
      busy : Bool;
      req : Bool;
      IEC_Timer_0_Instance : TON_TIME;
      tt : Int;
   END_VAR
   VAR_TEMP   // added for the SCL form of the ladder/FBD networks
      _w1 : Bool;
   END_VAR
BEGIN

REGION Network 1
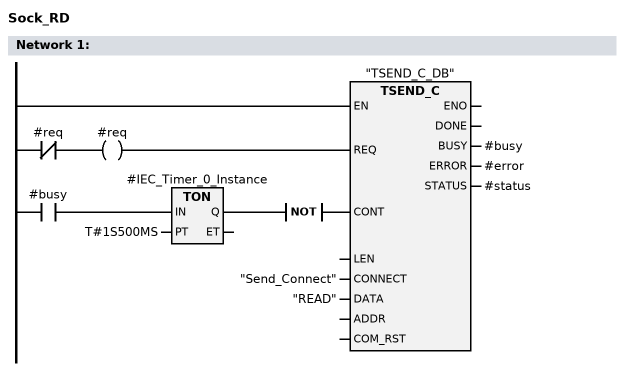
   #_w1 := NOT #req;
   #req := #_w1;
   #IEC_Timer_0_Instance(IN := #busy, PT := T#1S500MS);   // TON
   "TSEND_C_DB"(REQ := #_w1,   // TSEND_C
                CONT := NOT #IEC_Timer_0_Instance.Q,
                CONNECT := "Send_Connect",
                DATA := "READ",
                BUSY => #busy,
                ERROR => #error,
                STATUS => #status);
END_REGION
END_FUNCTION_BLOCK

// folder: Socket_Write

FUNCTION_BLOCK "Sock_WR"   // FB13, LAD
{ S7_Optimized_Access := 'TRUE' }
VERSION : 0.1
   VAR_OUTPUT
      error : Bool;
      stat : Word;
   END_VAR
   VAR
      busyTrcv : Bool;
      fall0 : Bool;
      IEC_Timer_0_Instance_0 : TON_TIME;
      IEC_Timer_0_Instance : TON_TIME;
      IEC_Timer_0_Instance_1 : TOF_TIME;
      TRCV_C_Instance : TRCV_C;
   END_VAR
   VAR_TEMP
      "upper.width_err" : Bool;
      "upper.delay_err" : Bool;
      "upper.speed_err" : Bool;
      "upper.speedJog_err" : Bool;
      "upper.speedInitia_err" : Bool;
      "upper.pulsesPerMeter_err" : Bool;
      "upper.offsetCenter_err" : Bool;
      "lower.width_err" : Bool;
      "lower.delay_err" : Bool;
      "lower.speed_err" : Bool;
      "lower.speedJog_err" : Bool;
      "lower.speedInitia_err" : Bool;
      "lower.pulsesPerMeter_err" : Bool;
      "lower.offsetCenter_err" : Bool;
      enyValueError : Bool;
      first_start : Bool;
   END_VAR
   VAR_TEMP   // added for the SCL form of the ladder/FBD networks
      _w1 : Bool;
   END_VAR
BEGIN

REGION Network 1
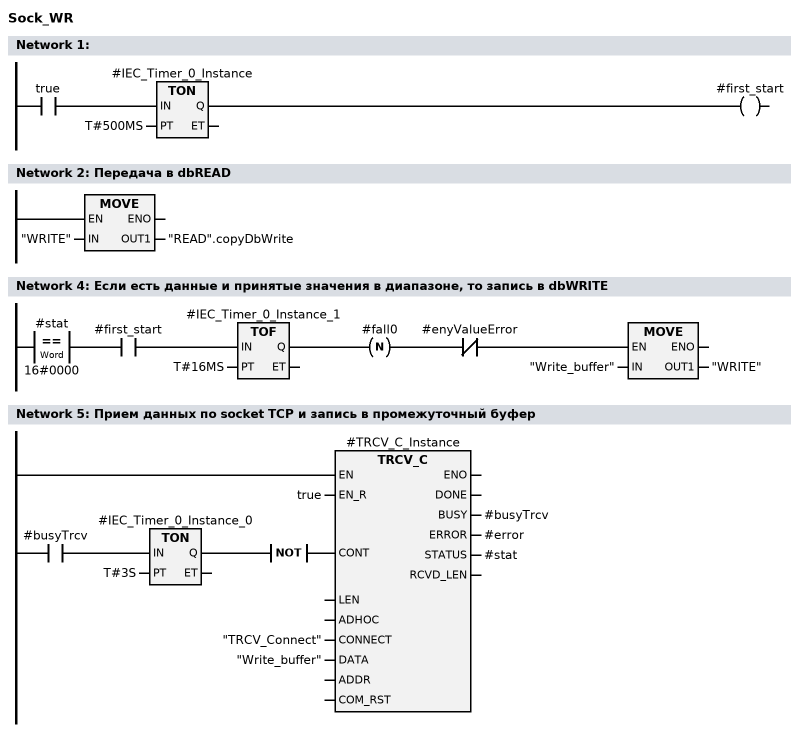
   #IEC_Timer_0_Instance(IN := true, PT := T#500MS);   // TON
   #first_start := #IEC_Timer_0_Instance.Q;
END_REGION

REGION Network 2: Передача в dbREAD
   RUNG wire#powerrail
      Move(in := "WRITE", out1 => "READ".copyDbWrite)
   END_RUNG
   // the same network as SCL:
   "READ".copyDbWrite := "WRITE";
END_REGION

REGION Network 3 (SCL): Проверка принятых числел, входят ли они в диапазон
   // Для верхнего
   IF ("Write_buffer".upper.width < 100) OR ("Write_buffer".upper.width > 2582) THEN
       #"upper.width_err" := true;
   ELSIF ("Write_buffer".upper.delay < 0) OR ("Write_buffer".upper.delay > 100_000) THEN
       #"upper.delay_err" := true;
   ELSIF ("Write_buffer".upper.speed < 1) OR ("Write_buffer".upper.speed > 100) THEN
       #"upper.speed_err" := true;
   ELSIF ("Write_buffer".upper.speedJog < 1) OR ("Write_buffer".upper.speedJog > 100) THEN
       #"upper.speedJog_err" := true;
   ELSIF ("Write_buffer".upper.speedInitia < 1) OR ("Write_buffer".upper.speedInitia > 100) THEN
       #"upper.speedInitia_err" := true;
   ELSIF ("Write_buffer".upper.pulsesPerMeter < 1) OR ("Write_buffer".upper.pulsesPerMeter > 10_000_000) THEN
       #"upper.pulsesPerMeter_err" := true;
   ELSIF ("Write_buffer".upper.offsetCenter < -1290) OR ("Write_buffer".upper.offsetCenter > 1291) THEN
       #"upper.offsetCenter_err" := true;
   END_IF;

   // Для нижнего
   IF ("Write_buffer".lower.width < 100) OR ("Write_buffer".lower.width > 2582) THEN
       #"lower.width_err" := true;
   ELSIF ("Write_buffer".lower.delay < 0) OR ("Write_buffer".lower.delay > 100_000) THEN
       #"lower.delay_err" := true;
   ELSIF ("Write_buffer".lower.speed < 1) OR ("Write_buffer".lower.speed > 100) THEN
       #"lower.speed_err" := true;
   ELSIF ("Write_buffer".lower.speedJog < 1) OR ("Write_buffer".lower.speedJog > 100) THEN
       #"lower.speedJog_err" := true;
   ELSIF ("Write_buffer".lower.speedInitia < 1) OR ("Write_buffer".lower.speedInitia > 100) THEN
       #"lower.speedInitia_err" := true;
   ELSIF ("Write_buffer".lower.pulsesPerMeter < 1) OR ("Write_buffer".lower.pulsesPerMeter > 10_000_000) THEN
       #"lower.pulsesPerMeter_err" := true;
   ELSIF ("Write_buffer".lower.offsetCenter < -1290) OR ("Write_buffer".lower.offsetCenter > 1291) THEN
       #"lower.offsetCenter_err" := true;
   END_IF;

   // Флаг если хотя бы одна переменная вышла за диапазон.
   #enyValueError := (
       #"upper.width_err" OR
       #"upper.delay_err" OR
       #"upper.speed_err" OR
       #"upper.speedJog_err" OR
       #"upper.speedInitia_err" OR
       #"upper.pulsesPerMeter_err" OR
       #"upper.offsetCenter_err" OR
       #"lower.width_err" OR
       #"lower.delay_err" OR
       #"lower.speed_err" OR
       #"lower.speedJog_err" OR
       #"lower.speedInitia_err" OR
       #"lower.pulsesPerMeter_err" OR
       #"lower.offsetCenter_err"
   );
END_REGION

REGION Network 4: Если есть данные и принятые значения в диапазоне, то запись в dbWRITE
   #IEC_Timer_0_Instance_1(IN := (#stat = 16#0000) AND #first_start, PT := T#16MS);   // TOF
   #_w1 := NOT #IEC_Timer_0_Instance_1.Q AND #fall0;   // falling edge
   #fall0 := #IEC_Timer_0_Instance_1.Q;
   IF #_w1 AND NOT #enyValueError THEN "WRITE" := "Write_buffer"; END_IF;
END_REGION

REGION Network 5: Прием данных по socket TCP и запись в промежуточный буфер
   #IEC_Timer_0_Instance_0(IN := #busyTrcv, PT := T#3S);   // TON
   #TRCV_C_Instance(EN_R := true,   // TRCV_C
                    CONT := NOT #IEC_Timer_0_Instance_0.Q,
                    CONNECT := "TRCV_Connect",
                    DATA := "Write_buffer",
                    BUSY => #busyTrcv,
                    ERROR => #error,
                    STATUS => #stat);
END_REGION
END_FUNCTION_BLOCK

// folder: functions

FUNCTION "binToDec" : Void   // FC1, SCL
{ S7_Optimized_Access := 'TRUE' }
VERSION : 0.1
   VAR_INPUT
      in0 : Bool;
      in1 : Bool;
   END_VAR
   VAR_OUTPUT
      out : USInt;
   END_VAR
BEGIN
   #out := 0;
   IF #in0 THEN
       #out := #out + 1;
   END_IF;

   IF #in1 THEN
       #out := #out + 2;
   END_IF;
END_FUNCTION

FUNCTION "bool4Coder" : Void   // FC6, SCL
{ S7_Optimized_Access := 'TRUE' }
VERSION : 0.1
   VAR_INPUT
      in0 : Bool;
      in1 : Bool;
      in2 : Bool;
      in3 : Bool;
   END_VAR
   VAR_OUTPUT
      out : USInt;
   END_VAR
BEGIN
   IF #in0 THEN
       #out := 1;
   END_IF;

   IF #in1 THEN
       #out := 2;
   END_IF;

   IF #in2 THEN
       #out := 3;
   END_IF;

   IF #in3 THEN
       #out := 4;
   END_IF;
END_FUNCTION

FUNCTION "inputEdit" : Void   // FC7, SCL
{ S7_Optimized_Access := 'TRUE' }
VERSION : 0.1
   VAR_INPUT
      in0 : Bool;
      in0Edit : USInt;
      in1 : Bool;
      in1Edit : USInt;
      in2 : Bool;
      in2Edit : USInt;
      in3 : Bool;
      in3Edit : USInt;
      in4 : Bool;
      in4Edit : USInt;
      in5 : Bool;
      in5Edit : USInt;
      in6 : Bool;
      in6Edit : USInt;
      in7 : Bool;
      in7Edit : USInt;
      in8 : Bool;
      in8Edit : USInt;
      in9 : Bool;
      in9Edit : USInt;
      in10 : Bool;
      in10Edit : USInt;
   END_VAR
   VAR_OUTPUT
      out0 : Bool;
      out1 : Bool;
      out2 : Bool;
      out3 : Bool;
      out4 : Bool;
      out5 : Bool;
      out6 : Bool;
      out7 : Bool;
      out8 : Bool;
      out9 : Bool;
      out10 : Bool;
   END_VAR
BEGIN

   IF #in0Edit = 0 THEN
       #out0 := #in0;
   ELSIF #in0Edit = 1 THEN
       #out0 := FALSE;
   ELSIF #in0Edit = 2 THEN
       #out0 := TRUE;
   ELSE
       #out0 := #in0;
   END_IF;

   IF #in1Edit = 0 THEN
       #out1 := #in0;
   ELSIF #in1Edit = 1 THEN
       #out1 := FALSE;
   ELSIF #in1Edit = 2 THEN
       #out1 := TRUE;
   ELSE
       #out1 := #in0;
   END_IF;

   IF #in2Edit = 0 THEN
       #out2 := #in0;
   ELSIF #in2Edit = 1 THEN
       #out2 := FALSE;
   ELSIF #in2Edit = 2 THEN
       #out2 := TRUE;
   ELSE
       #out2 := #in0;
   END_IF;

   IF #in3Edit = 0 THEN
       #out3 := #in0;
   ELSIF #in3Edit = 1 THEN
       #out3 := FALSE;
   ELSIF #in3Edit = 2 THEN
       #out3 := TRUE;
   ELSE
       #out3 := #in0;
   END_IF;

   IF #in4Edit = 0 THEN
       #out4 := #in0;
   ELSIF #in0Edit = 1 THEN
       #out4 := FALSE;
   ELSIF #in0Edit = 2 THEN
       #out4 := TRUE;
   ELSE
       #out4 := #in0;
   END_IF;

   IF #in5Edit = 0 THEN
       #out5 := #in0;
   ELSIF #in4Edit = 1 THEN
       #out5 := FALSE;
   ELSIF #in4Edit = 2 THEN
       #out5 := TRUE;
   ELSE
       #out5 := #in0;
   END_IF;

   IF #in6Edit = 0 THEN
       #out6 := #in0;
   ELSIF #in6Edit = 1 THEN
       #out6 := FALSE;
   ELSIF #in6Edit = 2 THEN
       #out6 := TRUE;
   ELSE
       #out6 := #in0;
   END_IF;

   IF #in7Edit = 0 THEN
       #out7 := #in0;
   ELSIF #in7Edit = 1 THEN
       #out7 := FALSE;
   ELSIF #in7Edit = 2 THEN
       #out7 := TRUE;
   ELSE
       #out7 := #in0;
   END_IF;

   IF #in8Edit = 0 THEN
       #out8 := #in0;
   ELSIF #in8Edit = 1 THEN
       #out8 := FALSE;
   ELSIF #in8Edit = 2 THEN
       #out8 := TRUE;
   ELSE
       #out8 := #in0;
   END_IF;

   IF #in9Edit = 0 THEN
       #out9 := #in0;
   ELSIF #in9Edit = 1 THEN
       #out9 := FALSE;
   ELSIF #in9Edit = 2 THEN
       #out9 := TRUE;
   ELSE
       #out9 := #in0;
   END_IF;

   IF #in10Edit = 0 THEN
       #out10 := #in0;
   ELSIF #in10Edit = 1 THEN
       #out10 := FALSE;
   ELSIF #in10Edit = 2 THEN
       #out10 := TRUE;
   ELSE
       #out10 := #in0;
   END_IF;
END_FUNCTION

// folder: initializing

FUNCTION_BLOCK "initializing"   // FB2, LAD
{ S7_Optimized_Access := 'TRUE' }
VERSION : 0.1
   VAR_INPUT
      emergencyStop : Bool;   // Аварийный стоп
      driveAlarm : Bool;   // Авария драйвера шагового двигателя
      mode : Bool;   // Режим (Авто - true)
      SW1 : Bool;   // Концевик - 1
      SW2 : Bool;   // Концевик - 2
      "^changeDist1" : Bool;   // Импульс если изменилось число L1
      "^changeDist2" : Bool := false;   // Импульс если изменилось число L2
      modeRun : Bool;   // Флаг режима Работа (автоматическое перемещение)
      speedInitia : DInt;   // Скорость перемещения при инициализации (имп/сек)
      speedManual : DInt;   // Скорость перемещения в ручном режиме (имп/сек)
   END_VAR
   VAR_OUTPUT
      modeInitia : Bool;   // Статус - идет инициализация
      initializing : Bool;   // Флаг - инициализация
      initialOKdelay : Bool;   // Инициализация завершена (с запазданием)
      initialOK : Bool;   // Инициализация завершена (без задержки)
      speedJog : DInt;   // Скорость для блока "Move_Jog" (имп/сек)
   END_VAR
   VAR
      "^SW2Up" : Bool;
      triggInitiaUp : Bool;
      initializingUp : Bool;
      "^initiaUpOk" : Bool;
      triggUpOk : Bool;
      raise0 : Bool;
      raise1 : Bool := false;
      raise2 : Bool := false;
      raise3 : Bool := false;
      raise4 : Bool := false;
      IEC_Timer_0_Instance : TON_TIME;
      IEC_Timer_0_Instance_1 : TOF_TIME;
      IEC_Timer_0_Instance_2 : TON_TIME;
      IEC_Timer_0_Instance_3 : TON_TIME;
      IEC_Timer_0_Instance_4 : TOF_TIME;
      IEC_Timer_0_Instance_5 : TOF_TIME;
      IEC_Timer_0_Instance_6 : TON_TIME;
      IEC_Timer_0_Instance_7 : TOF_TIME;
      IEC_Timer_0_Instance_8 : TOF_TIME;
      IEC_Timer_0_Instance_10 : TON_TIME;
      IEC_Timer_0_Instance_11 : TOF_TIME;
   END_VAR
   VAR_TEMP
      enInitia : Bool;
      "^SW1Run" : Bool;
      reInitia0 : Bool;
      reInitia1 : Bool;
   END_VAR
   VAR_TEMP   // added for the SCL form of the ladder/FBD networks
      _w1 : Bool;
   END_VAR
BEGIN

REGION Network 1: Переключение на скорость при инициализации (верхнего)
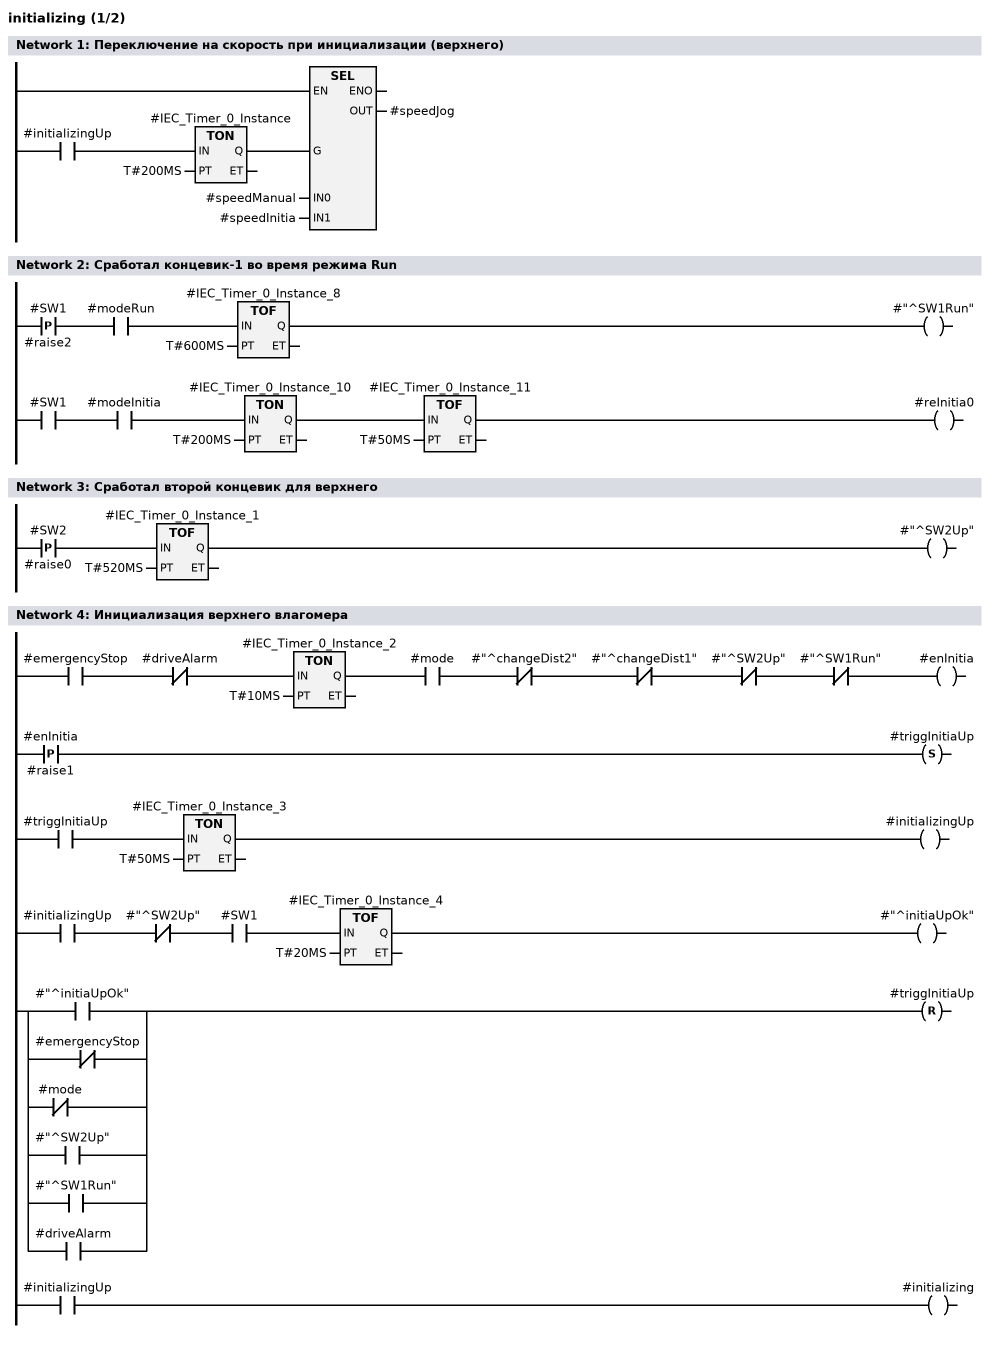
   #IEC_Timer_0_Instance(IN := #initializingUp, PT := T#200MS);   // TON
   #speedJog := SEL(G := #IEC_Timer_0_Instance.Q, IN0 := #speedManual, IN1 := #speedInitia);
END_REGION

REGION Network 2: Сработал концевик-1 во время режима Run
   #_w1 := #SW1 AND NOT #raise2;   // rising edge of #SW1
   #raise2 := #SW1;
   #IEC_Timer_0_Instance_8(IN := #_w1 AND #modeRun, PT := T#600MS);   // TOF
   #"^SW1Run" := #IEC_Timer_0_Instance_8.Q;
   #IEC_Timer_0_Instance_10(IN := #SW1 AND #modeInitia, PT := T#200MS);   // TON
   #IEC_Timer_0_Instance_11(IN := #IEC_Timer_0_Instance_10.Q, PT := T#50MS);   // TOF
   #reInitia0 := #IEC_Timer_0_Instance_11.Q;
END_REGION

REGION Network 3: Сработал второй концевик для верхнего
   #_w1 := #SW2 AND NOT #raise0;   // rising edge of #SW2
   #raise0 := #SW2;
   #IEC_Timer_0_Instance_1(IN := #_w1, PT := T#520MS);   // TOF
   #"^SW2Up" := #IEC_Timer_0_Instance_1.Q;
END_REGION

REGION Network 4: Инициализация верхнего влагомера
   #IEC_Timer_0_Instance_2(IN := #emergencyStop AND NOT #driveAlarm, PT := T#10MS);   // TON
   #enInitia := #IEC_Timer_0_Instance_2.Q AND #mode AND NOT #"^changeDist2" AND NOT #"^changeDist1" AND NOT #"^SW2Up" AND NOT #"^SW1Run";
   #_w1 := #enInitia AND NOT #raise1;   // rising edge of #enInitia
   #raise1 := #enInitia;
   IF #_w1 THEN #triggInitiaUp := TRUE; END_IF;
   #IEC_Timer_0_Instance_3(IN := #triggInitiaUp, PT := T#50MS);   // TON
   #initializingUp := #IEC_Timer_0_Instance_3.Q;
   #IEC_Timer_0_Instance_4(IN := #initializingUp AND NOT #"^SW2Up" AND #SW1, PT := T#20MS);   // TOF
   #"^initiaUpOk" := #IEC_Timer_0_Instance_4.Q;
   IF #"^initiaUpOk" OR NOT #emergencyStop OR NOT #mode OR #"^SW2Up" OR #"^SW1Run" OR #driveAlarm THEN
       #triggInitiaUp := FALSE;
   END_IF;
   #initializing := #initializingUp;
END_REGION

REGION Network 5: Инициализация верхнего прошла успешно
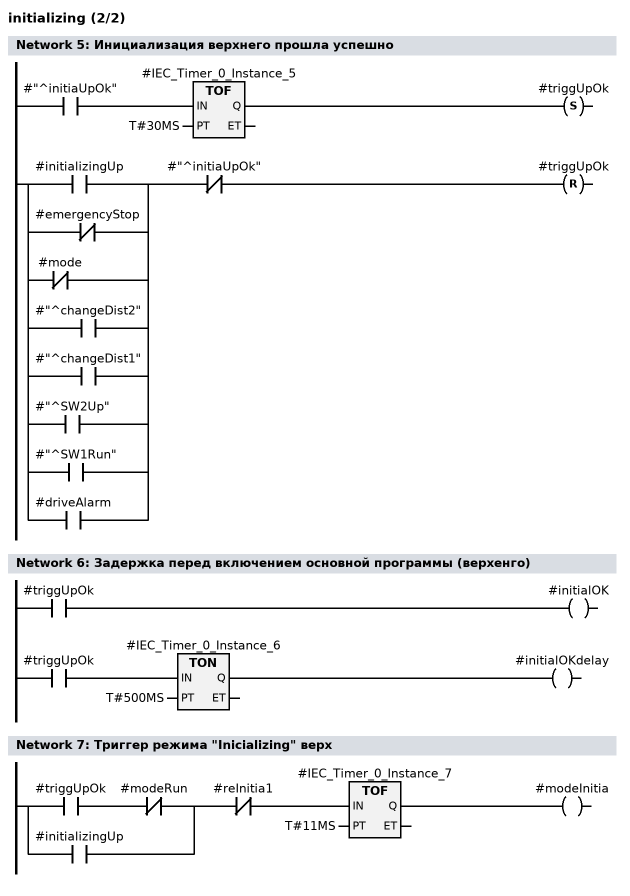
   #IEC_Timer_0_Instance_5(IN := #"^initiaUpOk", PT := T#30MS);   // TOF
   IF #IEC_Timer_0_Instance_5.Q THEN #triggUpOk := TRUE; END_IF;
   IF (#initializingUp OR NOT #emergencyStop OR NOT #mode OR #"^changeDist2" OR #"^changeDist1" OR #"^SW2Up" OR #"^SW1Run" OR #driveAlarm) AND NOT #"^initiaUpOk" THEN
       #triggUpOk := FALSE;
   END_IF;
END_REGION

REGION Network 6: Задержка перед включением основной программы (верхенго)
   #initialOK := #triggUpOk;
   #IEC_Timer_0_Instance_6(IN := #triggUpOk, PT := T#500MS);   // TON
   #initialOKdelay := #IEC_Timer_0_Instance_6.Q;
END_REGION

REGION Network 7: Триггер режимa "Inicializing" верх
   #IEC_Timer_0_Instance_7(IN := ((#triggUpOk AND NOT #modeRun) OR #initializingUp) AND NOT #reInitia1,   // TOF
                           PT := T#11MS);
   #modeInitia := #IEC_Timer_0_Instance_7.Q;
END_REGION
END_FUNCTION_BLOCK

// folder: math

FUNCTION_BLOCK "math"   // FB7, LAD
{ S7_Optimized_Access := 'TRUE' }
VERSION : 0.1
   VAR_INPUT
      modeRunUp : Bool;   // Статус - активно авто перемещение (верх)
      modeRunDown : Bool;   // Статус - активно авто перемещение (Низ)
      directionUp : Bool;   // Направление движения (верх)
      directionDown : Bool;   // Направление движения (Низ)
      L2UpMM : DInt;   // ширина обЪекта измерения (верх), мм
      L2DownMM : DInt;   // ширина обЪекта измерения (Низ), мм
      adjustL1Up : DInt;   // коррекция длины L1 (верх)
      adjustL1Down : DInt;   // коррекция длины L1 (Низ)
      pulsesPerMeterUp : DInt;   // Уставка - кол-во импульсов на 1 метр пути (верх)
      pulsesPerMeterDown : DInt;   // Уставка - кол-во импульсов на 1 метр пути (Низ)
      speedUp : DInt;   // Скорость в режиме авто (верх), %
      speedDown : DInt;   // Скорость в режиме авто (Низ), %
      speedInitiaUp : DInt;   // Скорость при инициализации (верх), %
      speedInitiaDown : DInt;   // Скорость при инициализации (Низ), %
      speedJogUp : DInt;   // Скорость в ручном режиме (верх), %
      speedJogDown : DInt;   // Скорость в ручном режиме (Низ), %
   END_VAR
   VAR_OUTPUT
      L1UpMM : DInt;   // расстояние от нулевой позиции до начала обЪекта измерения (верх), мм
      L1DownMM : DInt;   // расстояние от нулевой позиции до начала обЪекта измерения (Низ), мм
      pulsesPerMMUp : DInt;   // Вычисленное кол-во импульсов на 1мм пути (верх)
      pulsesPerMMDown : DInt;   // Вычисленное кол-во импульсов на 1мм пути (Низ)
      setPulsesUp : DInt;   // Текущая уставка длины L (верх)
      setPulsesDown : DInt;   // Текущая уставка длины L (Низ)
      actualPulsesUp : DInt;   // Текущая уставка длины L с инверсией знака для обратного движения (верх)
      actualPulsesDown : DInt;   // Текущая уставка длины L с инверсией знака для обратного движения (Низ)
      speedPulsesUp : DInt;   // Скорость перемещения в режиме авто (имп/сек) верх
      speedPulsesDown : DInt;   // Скорость перемещения в режиме авто (имп/сек) Низ
      speedPulsesIniUp : DInt;   // Скорость перемещения при инициализации (имп/сек) верх
      speedPulsesIniDown : DInt;   // Скорость перемещения при инициализации (имп/сек) Низ
      speedPulsesJogUp : DInt;   // Скорость перемещения в ручном режиме (имп/сек) верх
      speedPulsesJogDown : DInt;   // Скорость перемещения в ручном режиме (имп/сек) Низ
      "^ChangeL1Up" : Bool;   // Импульс если изменилось число L1 (верх)
      "^ChangeL2Up" : Bool;   // Импульс если изменилось число L2 (верх)
      "^ChangeL1Down" : Bool;   // Импульс если изменилось число L1 (Низ)
      "^ChangeL2Down" : Bool;   // Импульс если изменилось число L2 (Низ)
   END_VAR
   VAR
      L1CalcUp : DInt;
      L1CalcDown : DInt;
      CurrLUp : DInt;
      CurrLDown : DInt;
      invPulsesUp : DInt;
      invPulsesDown : DInt;
      "^Ch_Dint_Instance" : "^Ch_Dint";
      "^Ch_Dint_Instance_1" : "^Ch_Dint";
      "^Ch_Dint_Instance_2" : "^Ch_Dint";
      "^Ch_Dint_Instance_3" : "^Ch_Dint";
   END_VAR
BEGIN

REGION Network 1 (SCL): расстояние от нулевой позиции до начала обЪекта измерения (верх), мм
   #L1CalcUp := (2582 - LIMIT(MN := 100, IN := #L2UpMM, MX := 2400)) / 2;
   #L1UpMM := #L1CalcUp + #adjustL1Up;

   #L1CalcDown := (2582 - LIMIT(MN := 100, IN := #L2DownMM, MX := 2400)) / 2;
   #L1DownMM := #L1CalcDown + #adjustL1Down;
END_REGION

REGION Network 2: Переключение L, пересчет с мм в импульсы, (верхний)
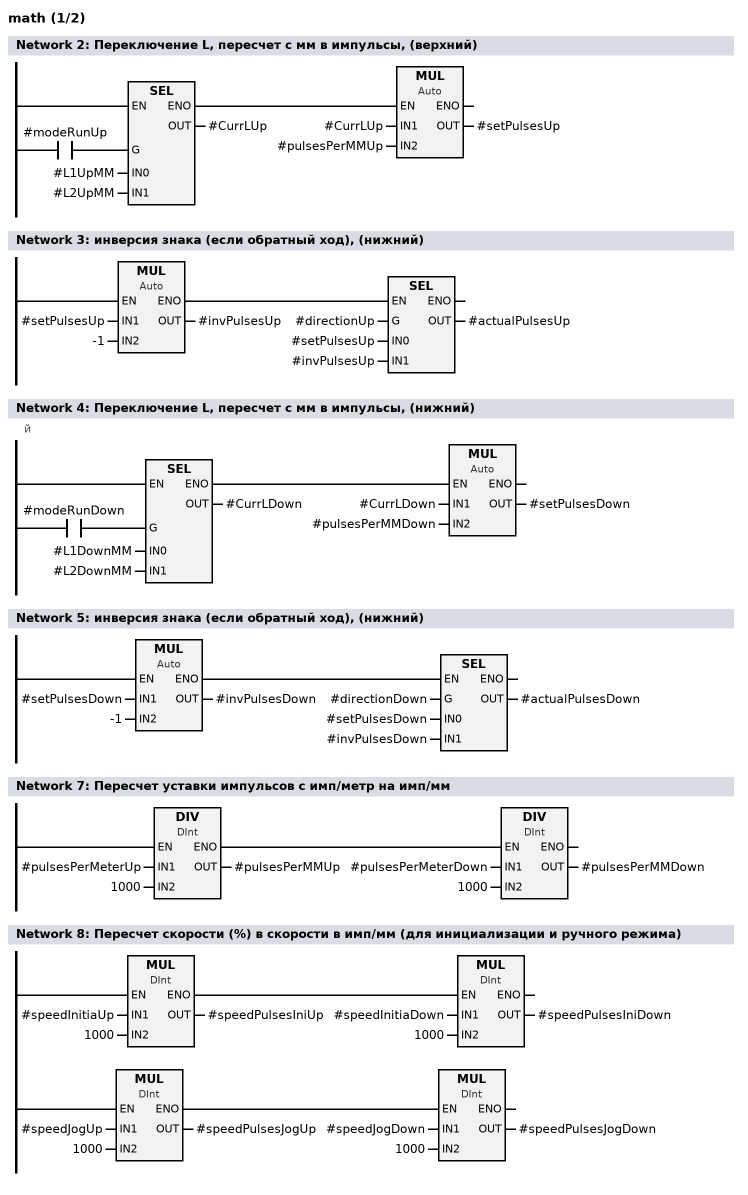
   // ENO of a box is taken as its EN; it also drops when the box reports an error
   #CurrLUp := SEL(G := #modeRunUp, IN0 := #L1UpMM, IN1 := #L2UpMM);
   #setPulsesUp := #CurrLUp * #pulsesPerMMUp;
END_REGION

REGION Network 3: инверсия знака (если обратный ход), (нижний)
   #invPulsesUp := #setPulsesUp * (-1);
   #actualPulsesUp := SEL(G := #directionUp, IN0 := #setPulsesUp, IN1 := #invPulsesUp);
END_REGION

REGION Network 4: Переключение L, пересчет с мм в импульсы, (нижний)
   // й
   // ENO of a box is taken as its EN; it also drops when the box reports an error
   #CurrLDown := SEL(G := #modeRunDown, IN0 := #L1DownMM, IN1 := #L2DownMM);
   #setPulsesDown := #CurrLDown * #pulsesPerMMDown;
END_REGION

REGION Network 5: инверсия знака (если обратный ход), (нижний)
   #invPulsesDown := #setPulsesDown * (-1);
   #actualPulsesDown := SEL(G := #directionDown, IN0 := #setPulsesDown, IN1 := #invPulsesDown);
END_REGION

REGION Network 6 (SCL): Пересчет скорости c %, в имп/сек (верх и низ)
   #speedPulsesUp := LIMIT(MN := 1, IN := #speedUp, MX := 100) * 720;
   #speedPulsesDown := LIMIT(MN := 1, IN := #speedDown, MX := 100) * 720;
END_REGION

REGION Network 7: Пересчет уставки импульсов с имп/метр на имп/мм
   RUNG wire#powerrail
      { S7_Templates := "SrcType := DInt" } Div(in1 := #pulsesPerMeterUp, in2 := 1000, out => #pulsesPerMMUp)
      { S7_Templates := "SrcType := DInt" } Div(in1 := #pulsesPerMeterDown, in2 := 1000, out => #pulsesPerMMDown)
   END_RUNG
   // the same network as SCL:
   #pulsesPerMMUp := #pulsesPerMeterUp / 1000;
   #pulsesPerMMDown := #pulsesPerMeterDown / 1000;
END_REGION

REGION Network 8: Пересчет скорости (%) в скорости в имп/мм (для инициализации и ручного режима)
   RUNG wire#powerrail
      { S7_Templates := "SrcType := DInt" } Mul(in1 := #speedInitiaUp, in2 := 1000, out => #speedPulsesIniUp)
      { S7_Templates := "SrcType := DInt" } Mul(in1 := #speedInitiaDown, in2 := 1000, out => #speedPulsesIniDown)
   END_RUNG
   RUNG wire#powerrail
      { S7_Templates := "SrcType := DInt" } Mul(in1 := #speedJogUp, in2 := 1000, out => #speedPulsesJogUp)
      { S7_Templates := "SrcType := DInt" } Mul(in1 := #speedJogDown, in2 := 1000, out => #speedPulsesJogDown)
   END_RUNG
   // the same network as SCL:
   #speedPulsesIniUp := #speedInitiaUp * 1000;
   #speedPulsesIniDown := #speedInitiaDown * 1000;
   #speedPulsesJogUp := #speedJogUp * 1000;
   #speedPulsesJogDown := #speedJogDown * 1000;
END_REGION

REGION Network 9: Импульс если была изменена уставка дистанции L
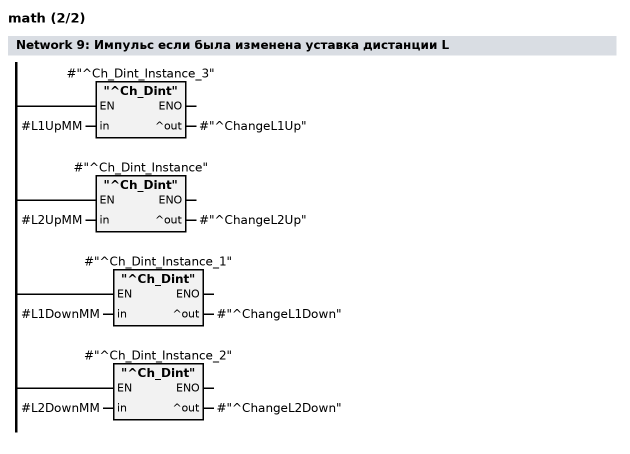
   RUNG wire#powerrail
      #"^Ch_Dint_Instance_3"(in := #L1UpMM, "^out" => #"^ChangeL1Up")
   END_RUNG
   RUNG wire#powerrail
      #"^Ch_Dint_Instance"(in := #L2UpMM, "^out" => #"^ChangeL2Up")
   END_RUNG
   RUNG wire#powerrail
      #"^Ch_Dint_Instance_1"(in := #L1DownMM, "^out" => #"^ChangeL1Down")
   END_RUNG
   RUNG wire#powerrail
      #"^Ch_Dint_Instance_2"(in := #L2DownMM, "^out" => #"^ChangeL2Down")
   END_RUNG
   // the same network as SCL:
   #"^Ch_Dint_Instance_3"(in := #L1UpMM, "^out" => #"^ChangeL1Up");   // "^Ch_Dint"
   #"^Ch_Dint_Instance"(in := #L2UpMM, "^out" => #"^ChangeL2Up");   // "^Ch_Dint"
   #"^Ch_Dint_Instance_1"(in := #L1DownMM, "^out" => #"^ChangeL1Down");   // "^Ch_Dint"
   #"^Ch_Dint_Instance_2"(in := #L2DownMM, "^out" => #"^ChangeL2Down");   // "^Ch_Dint"
END_REGION
END_FUNCTION_BLOCK

// folder: moving

FUNCTION_BLOCK "moving"   // FB5, LAD
{ S7_Optimized_Access := 'TRUE' }
VERSION : 0.1
   VAR_INPUT
      emergencyStop : Bool;   // Экстренный стоп
      initializing : Bool;   // Флаг - инициализация
      InitialOKdelay : Bool;   // Инициализация завершена (с запазданием)
      InitialOK : Bool;   // Инициализация завершена (без задержки)
      SW1 : Bool;   // Концевик - 1
      SW2 : Bool;   // Концевик - 2
      manualForward : Bool;   // Ручное перемещение вперед
      manualBackward : Bool;   // Ручное перемещение назад
      mode : Bool;   // Режим (Auto - true)
      delay : DInt;   // Задержка перед сменой направления движения, мс
      setPulses : DInt;   // Текущая уставка длины L
      pulsesPerMM : DInt;   // Вычисленное кол-во импульсов на 1мм пути
      speedPulses : DInt;   // Скорость перемещения в режиме авто (имп/сек)
      actualPulses : DInt;   // Текущая уставка длины L с инверсией знака. (Для обратного движения)
      speedJogPulses : DInt;   // Скорость перемещения в ручном режиме (имп/сек)
      axisDistance : Real;   // Текущий остаток импульсов до завершения позиционирования
      axisPower : TO_Axis;
      axisJog : TO_SpeedAxis;
      axisRelative : TO_PositioningAxis;
      enAxis : Bool;
   END_VAR
   VAR_OUTPUT
      driveDisable : Bool;   // Деактивация драйвера шагового двигателя
      backL2 : Bool;   // Флаг - обратное движение
      modeRun : Bool;   // Режим - работа (авто)
      currDistance : DInt;   // Текущее абсолютное положение на оси (на полотне измерения)
   END_VAR
   VAR
      IEC_Timer_0_Instance : TOF_TIME;
      IEC_Timer_0_Instance_1 : TOF_TIME;
      triggRunL1 : Bool;
      relativeDone : Bool;
      triggStartL2 : Bool;
      reStart : Bool;
      triggBackL2 : Bool;
      raiseFall0 : Bool;
      raiseFall1 : Bool := false;
      raiseFall2 : Bool := false;
      raiseFall3 : Bool := false;
      raiseFall4 : Bool := false;
      raiseFall5 : Bool := false;
      raiseFall6 : Bool := false;
      raiseFall7 : Bool := false;
      raiseFall8 : Bool := false;
      raiseFall9 : Bool;
      relativeStart : Bool;
      IEC_Timer_0_Instance_2 : TOF_TIME;
      IEC_Timer_0_Instance_3 : TOF_TIME;
      IEC_Timer_0_Instance_4 : TOF_TIME;
      IEC_Timer_0_Instance_5 : TOF_TIME;
      IEC_Timer_0_Instance_6 : TOF_TIME;
      CurrDistance_Instance_1 : "CurrDistance";
      MC_Power_Instance : MC_Power;
      MC_MoveJog_Instance : MC_MoveJog;
      MC_MoveRelative_Instance : MC_MoveRelative;
      IEC_Timer_0_Instance_9 : TOF_TIME;
      IEC_Timer_0_Instance_10 : TON_TIME;
      IEC_Timer_0_Instance_11 : TON_TIME;
      IEC_Timer_0_Instance_7 : TON_TIME;
      IEC_Timer_0_Instance_8 : TOF_TIME;
      IEC_Timer_0_Instance_12 : TON_TIME;
   END_VAR
   VAR_TEMP
      modeEn : Bool;
      L1toL2 : Bool;
      delayL2 : Bool;
      reDelayL2 : Bool;
      "^relativeStart" : Bool;
      onSW2 : Bool;
      jogForward : Bool;
      jogBackward : Bool;
   END_VAR
   VAR_TEMP   // added for the SCL form of the ladder/FBD networks
      _w1 : Bool;
      _w2 : Bool;
   END_VAR
BEGIN

REGION Network 1: деактивация оси, если сменился режим на "ручной"
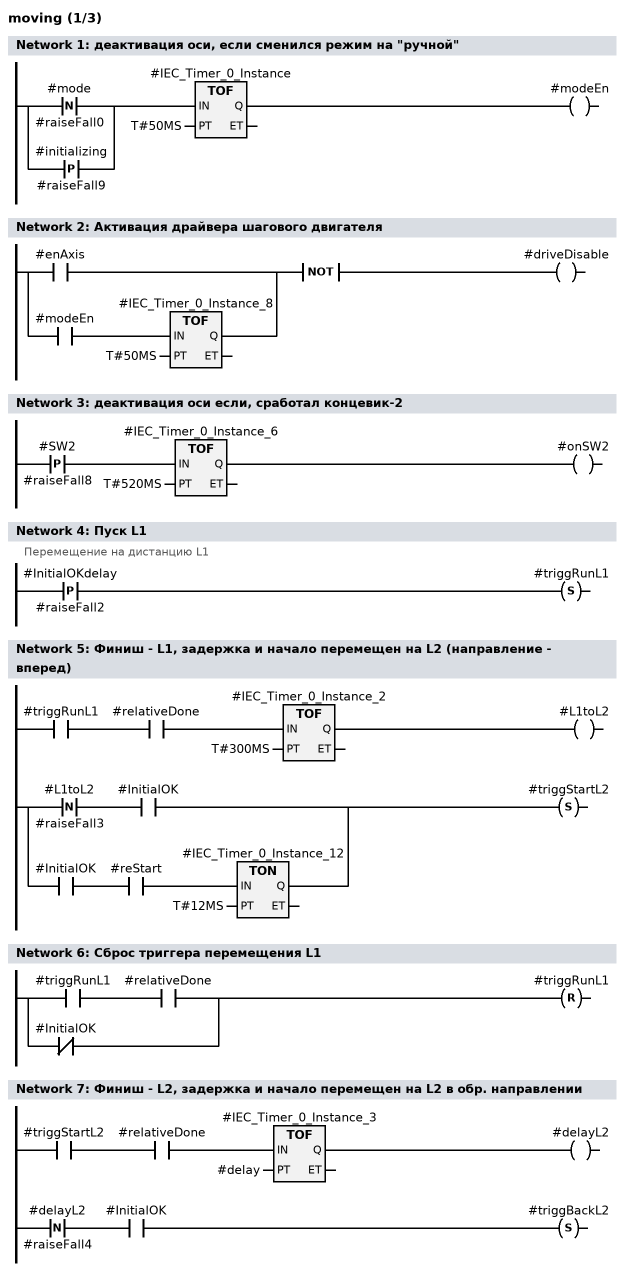
   #_w1 := NOT #mode AND #raiseFall0;   // falling edge of #mode
   #raiseFall0 := #mode;
   #_w2 := #initializing AND NOT #raiseFall9;   // rising edge of #initializing
   #raiseFall9 := #initializing;
   #IEC_Timer_0_Instance(IN := #_w1 OR #_w2, PT := T#50MS);   // TOF
   #modeEn := #IEC_Timer_0_Instance.Q;
END_REGION

REGION Network 2: Активация драйвера шагового двигателя
   #IEC_Timer_0_Instance_8(IN := #modeEn, PT := T#50MS);   // TOF
   #driveDisable := NOT (#enAxis OR #IEC_Timer_0_Instance_8.Q);
END_REGION

REGION Network 3: деактивация оси если, сработал концевик-2
   #_w1 := #SW2 AND NOT #raiseFall8;   // rising edge of #SW2
   #raiseFall8 := #SW2;
   #IEC_Timer_0_Instance_6(IN := #_w1, PT := T#520MS);   // TOF
   #onSW2 := #IEC_Timer_0_Instance_6.Q;
END_REGION

REGION Network 4: Пуск L1
   // Перемещение на дистанцию L1
   RUNG wire#powerrail
      P_Contact(operand := #InitialOKdelay, bit := #raiseFall2)
      S_Coil( #triggRunL1 )
   END_RUNG
   // the same network as SCL:
   #_w1 := #InitialOKdelay AND NOT #raiseFall2;   // rising edge of #InitialOKdelay
   #raiseFall2 := #InitialOKdelay;
   IF #_w1 THEN #triggRunL1 := TRUE; END_IF;
END_REGION

REGION Network 5: Финиш - L1, задержка и начало перемещен на L2 (направление - вперед)
   #IEC_Timer_0_Instance_2(IN := #triggRunL1 AND #relativeDone, PT := T#300MS);   // TOF
   #L1toL2 := #IEC_Timer_0_Instance_2.Q;
   #_w1 := NOT #L1toL2 AND #raiseFall3;   // falling edge of #L1toL2
   #raiseFall3 := #L1toL2;
   #IEC_Timer_0_Instance_12(IN := #InitialOK AND #reStart, PT := T#12MS);   // TON
   IF (#_w1 AND #InitialOK) OR #IEC_Timer_0_Instance_12.Q THEN #triggStartL2 := TRUE; END_IF;
END_REGION

REGION Network 6: Сброс триггера перемещения L1
   RUNG wire#powerrail
      Contact( #triggRunL1 )
      Contact( #relativeDone )
      wire#w1
      R_Coil( #triggRunL1 )
   END_RUNG
   RUNG wire#powerrail
      I_Contact( #InitialOK )
   END_RUNG wire#w1
   // the same network as SCL:
   IF (#triggRunL1 AND #relativeDone) OR NOT #InitialOK THEN #triggRunL1 := FALSE; END_IF;
END_REGION

REGION Network 7: Финиш - L2, задержка и начало перемещен на L2 в обр. направлении
   #IEC_Timer_0_Instance_3(IN := #triggStartL2 AND #relativeDone, PT := #delay);   // TOF
   #delayL2 := #IEC_Timer_0_Instance_3.Q;
   #_w1 := NOT #delayL2 AND #raiseFall4;   // falling edge of #delayL2
   #raiseFall4 := #delayL2;
   IF #_w1 AND #InitialOK THEN #triggBackL2 := TRUE; END_IF;
END_REGION

REGION Network 8: Сброс триггера перемещения L2 (направление - вперед)
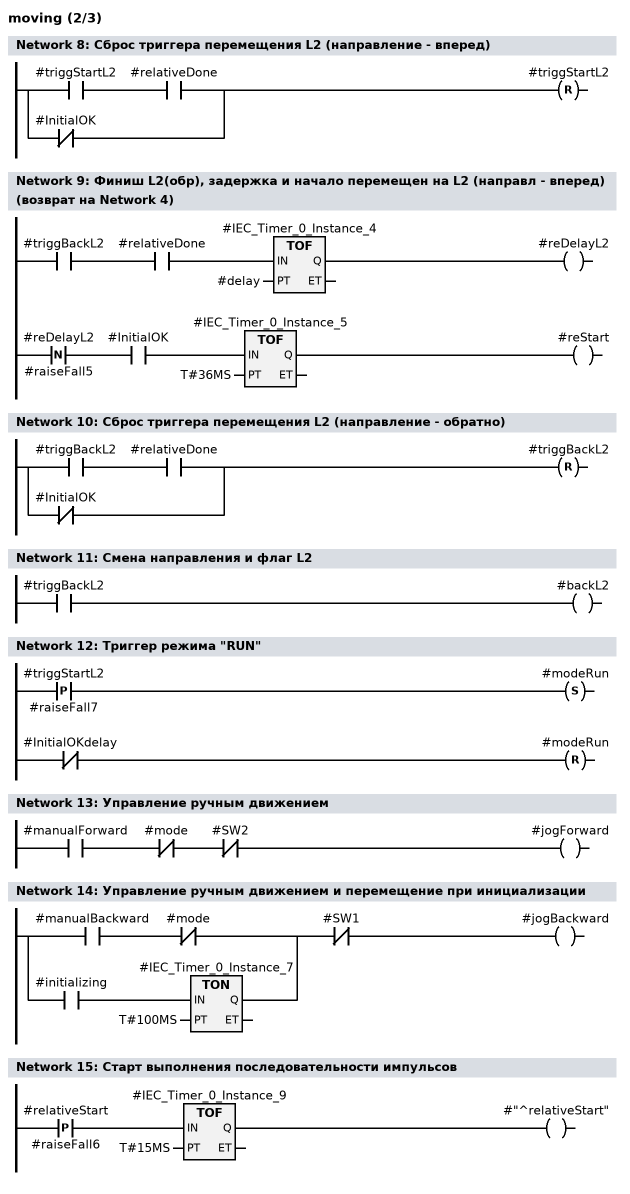
   RUNG wire#powerrail
      Contact( #triggStartL2 )
      Contact( #relativeDone )
      wire#w1
      R_Coil( #triggStartL2 )
   END_RUNG
   RUNG wire#powerrail
      I_Contact( #InitialOK )
   END_RUNG wire#w1
   // the same network as SCL:
   IF (#triggStartL2 AND #relativeDone) OR NOT #InitialOK THEN #triggStartL2 := FALSE; END_IF;
END_REGION

REGION Network 9: Финиш L2(обр), задержка и начало перемещен на L2 (направл - вперед) (возврат на Network 4)
   #IEC_Timer_0_Instance_4(IN := #triggBackL2 AND #relativeDone, PT := #delay);   // TOF
   #reDelayL2 := #IEC_Timer_0_Instance_4.Q;
   #_w1 := NOT #reDelayL2 AND #raiseFall5;   // falling edge of #reDelayL2
   #raiseFall5 := #reDelayL2;
   #IEC_Timer_0_Instance_5(IN := #_w1 AND #InitialOK, PT := T#36MS);   // TOF
   #reStart := #IEC_Timer_0_Instance_5.Q;
END_REGION

REGION Network 10: Сброс триггера перемещения L2 (направление - обратно)
   RUNG wire#powerrail
      Contact( #triggBackL2 )
      Contact( #relativeDone )
      wire#w1
      R_Coil( #triggBackL2 )
   END_RUNG
   RUNG wire#powerrail
      I_Contact( #InitialOK )
   END_RUNG wire#w1
   // the same network as SCL:
   IF (#triggBackL2 AND #relativeDone) OR NOT #InitialOK THEN #triggBackL2 := FALSE; END_IF;
END_REGION

REGION Network 11: Смена направления и флаг L2
   RUNG wire#powerrail
      Contact( #triggBackL2 )
      Coil( #backL2 )
   END_RUNG
   // the same network as SCL:
   #backL2 := #triggBackL2;
END_REGION

REGION Network 12: Триггер режимa "RUN"
   RUNG wire#powerrail
      P_Contact(operand := #triggStartL2, bit := #raiseFall7)
      S_Coil( #modeRun )
   END_RUNG
   RUNG wire#powerrail
      I_Contact( #InitialOKdelay )
      R_Coil( #modeRun )
   END_RUNG
   // the same network as SCL:
   #_w1 := #triggStartL2 AND NOT #raiseFall7;   // rising edge of #triggStartL2
   #raiseFall7 := #triggStartL2;
   IF #_w1 THEN #modeRun := TRUE; END_IF;
   IF NOT #InitialOKdelay THEN #modeRun := FALSE; END_IF;
END_REGION

REGION Network 13: Управление ручным движением
   RUNG wire#powerrail
      Contact( #manualForward )
      I_Contact( #mode )
      I_Contact( #SW2 )
      Coil( #jogForward )
   END_RUNG
   // the same network as SCL:
   #jogForward := #manualForward AND NOT #mode AND NOT #SW2;
END_REGION

REGION Network 14: Управление ручным движением и перемещение при инициализации
   #IEC_Timer_0_Instance_7(IN := #initializing, PT := T#100MS);   // TON
   #jogBackward := ((#manualBackward AND NOT #mode) OR #IEC_Timer_0_Instance_7.Q) AND NOT #SW1;
END_REGION

REGION Network 15: Cтарт выполнения последовательности импульсов
   #_w1 := #relativeStart AND NOT #raiseFall6;   // rising edge of #relativeStart
   #raiseFall6 := #relativeStart;
   #IEC_Timer_0_Instance_9(IN := #_w1, PT := T#15MS);   // TOF
   #"^relativeStart" := #IEC_Timer_0_Instance_9.Q;
END_REGION

REGION Network 16: Блоки Motion control
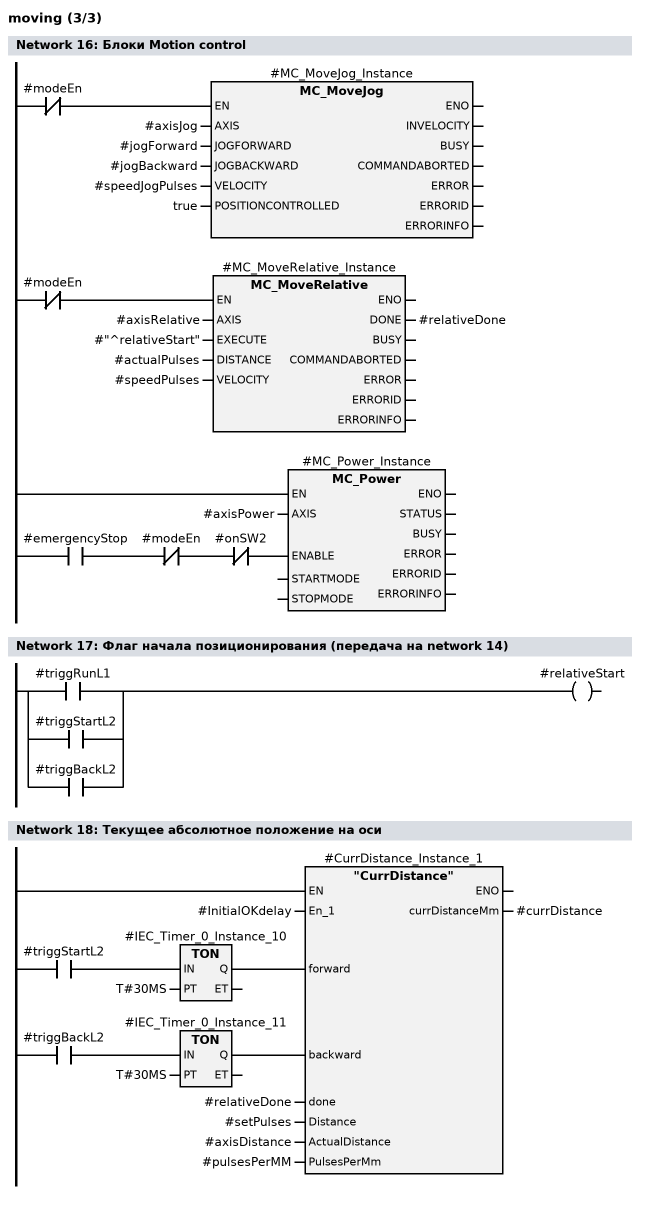
   IF NOT #modeEn THEN
       #MC_MoveJog_Instance(Axis := #axisJog,   // MC_MoveJog
                            JogForward := #jogForward,
                            JogBackward := #jogBackward,
                            Velocity := #speedJogPulses,
                            PositionControlled := true);
       #MC_MoveRelative_Instance(Axis := #axisRelative,   // MC_MoveRelative
                               Execute := #"^relativeStart",
                               Distance := #actualPulses,
                               Velocity := #speedPulses,
                               Done => #relativeDone);
   END_IF;
   #MC_Power_Instance(Axis := #axisPower, Enable := #emergencyStop AND NOT #modeEn AND NOT #onSW2);   // MC_Power
END_REGION

REGION Network 17: Флаг начала позиционирования (передача на network 14)
   RUNG wire#powerrail
      Contact( #triggRunL1 )
      wire#w1
      Coil( #relativeStart )
   END_RUNG
   RUNG wire#powerrail
      Contact( #triggStartL2 )
   END_RUNG wire#w1
   RUNG wire#powerrail
      Contact( #triggBackL2 )
   END_RUNG wire#w1
   // the same network as SCL:
   #relativeStart := #triggRunL1 OR #triggStartL2 OR #triggBackL2;
END_REGION

REGION Network 18: Текущее абсолютное положение на оси
   #IEC_Timer_0_Instance_10(IN := #triggStartL2, PT := T#30MS);   // TON
   #IEC_Timer_0_Instance_11(IN := #triggBackL2, PT := T#30MS);   // TON
   #CurrDistance_Instance_1(En_1 := #InitialOKdelay,   // "CurrDistance"
                           forward := #IEC_Timer_0_Instance_10.Q,
                           backward := #IEC_Timer_0_Instance_11.Q,
                           done := #relativeDone,
                           Distance := #setPulses,
                           ActualDistance := #axisDistance,
                           PulsesPerMm := #pulsesPerMM,
                           currDistanceMm => #currDistance);
END_REGION
END_FUNCTION_BLOCK

// folder: status&Mode

FUNCTION_BLOCK "statusMove"   // FB8, LAD
{ S7_Optimized_Access := 'TRUE' }
VERSION : 0.1
   VAR_INPUT
      emergStop : Bool;
      SW1Up : Bool;
      SW2Up : Bool;
      SW1Down : Bool;
      SW2Down : Bool;
      alarmDriveUp : Bool;
      alarmDriveDown : Bool;
      modeInitiaUp : Bool;
      modeInitiaDown : Bool;
      modeRunUp : Bool;
      modeRunDown : Bool;
      modeUp : Bool;
      modeDown : Bool;
      L1UpMMWrite : DInt;
      L2UpMMWrite : DInt;
      L1DownMMWrite : DInt;
      L2DownMMWrite : DInt;
      speedUpWrite : DInt;
      speedDownWrite : DInt;
   END_VAR
   VAR_OUTPUT
      modeUpRead : Bool;
      modeDownRead : Bool;
      L1UpMMRead : DInt;
      L2UpMMRead : DInt;
      L1DownMMRead : DInt;
      L2DownMMRead : DInt;
      speedUpRead : DInt;
      speedDownRead : DInt;
      statusUpHMI : USInt;
      statusDownHMI : USInt;
      statusUpRead : USInt;
      statusDownRead : USInt;
      modeUpDownHMI : USInt;
      statusGeneralHMI : USInt;
      SW1UpWrite : Bool;
      SW2UpWrite : Bool;
      SW1DownWrite : Bool;
      SW2DownWrite : Bool;
   END_VAR
BEGIN

REGION Network 1: Кодирование состояний программы (верх)
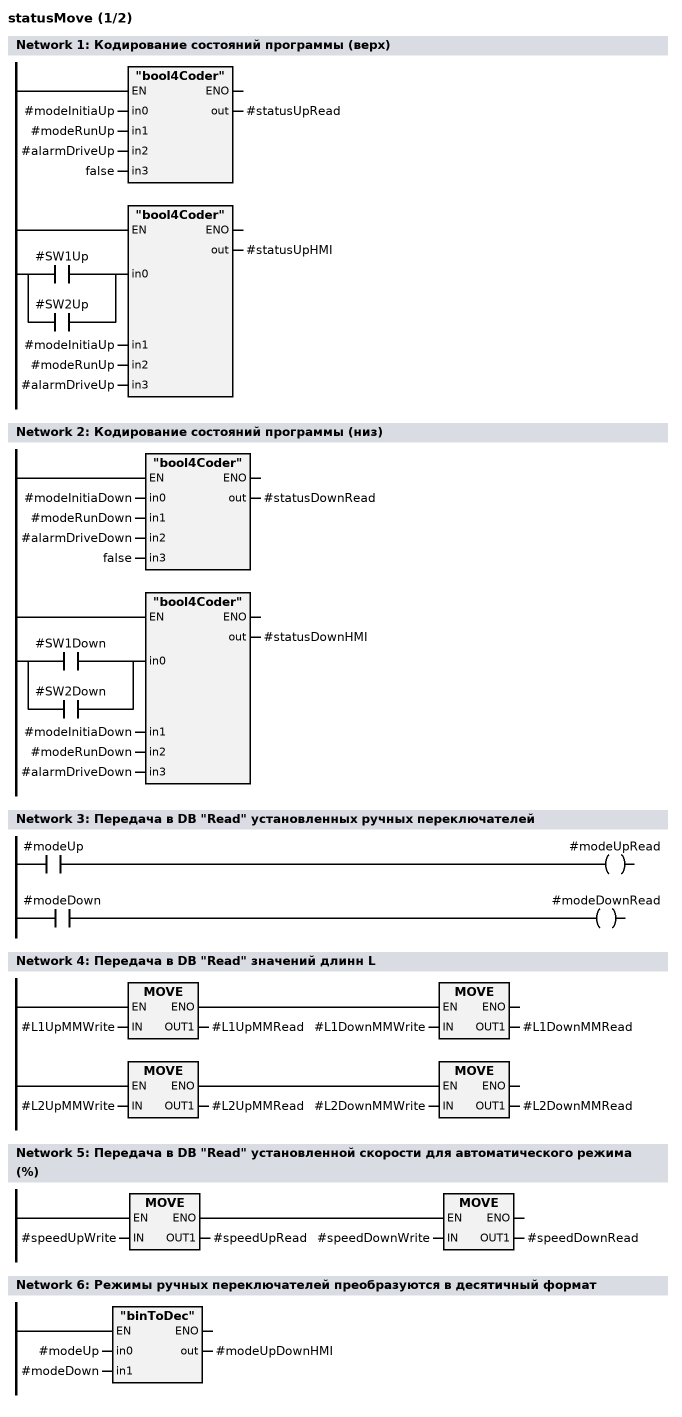
   RUNG wire#powerrail
      "bool4Coder"(in0 := #modeInitiaUp, in1 := #modeRunUp, in2 := #alarmDriveUp, in3 := false, out => #statusUpRead)
   END_RUNG
   RUNG wire#powerrail
      "bool4Coder"(in0 := wire#w1, in1 := #modeInitiaUp, in2 := #modeRunUp, in3 := #alarmDriveUp, out => #statusUpHMI)
   END_RUNG
   RUNG wire#powerrail
      Contact( #SW1Up )
   END_RUNG wire#w1
   RUNG wire#powerrail
      Contact( #SW2Up )
   END_RUNG wire#w1
   // the same network as SCL:
   "bool4Coder"(in0 := #modeInitiaUp,
                in1 := #modeRunUp,
                in2 := #alarmDriveUp,
                in3 := false,
                out => #statusUpRead);
   "bool4Coder"(in0 := #SW1Up OR #SW2Up,
                in1 := #modeInitiaUp,
                in2 := #modeRunUp,
                in3 := #alarmDriveUp,
                out => #statusUpHMI);
END_REGION

REGION Network 2: Кодирование состояний программы (низ)
   RUNG wire#powerrail
      "bool4Coder"(in0 := #modeInitiaDown, in1 := #modeRunDown, in2 := #alarmDriveDown, in3 := false, out => #statusDownRead)
   END_RUNG
   RUNG wire#powerrail
      "bool4Coder"(in0 := wire#w1, in1 := #modeInitiaDown, in2 := #modeRunDown, in3 := #alarmDriveDown, out => #statusDownHMI)
   END_RUNG
   RUNG wire#powerrail
      Contact( #SW1Down )
   END_RUNG wire#w1
   RUNG wire#powerrail
      Contact( #SW2Down )
   END_RUNG wire#w1
   // the same network as SCL:
   "bool4Coder"(in0 := #modeInitiaDown,
                in1 := #modeRunDown,
                in2 := #alarmDriveDown,
                in3 := false,
                out => #statusDownRead);
   "bool4Coder"(in0 := #SW1Down OR #SW2Down,
                in1 := #modeInitiaDown,
                in2 := #modeRunDown,
                in3 := #alarmDriveDown,
                out => #statusDownHMI);
END_REGION

REGION Network 3: Передача в DB "Read" установленных ручных переключателей
   RUNG wire#powerrail
      Contact( #modeUp )
      Coil( #modeUpRead )
   END_RUNG
   RUNG wire#powerrail
      Contact( #modeDown )
      Coil( #modeDownRead )
   END_RUNG
   // the same network as SCL:
   #modeUpRead := #modeUp;
   #modeDownRead := #modeDown;
END_REGION

REGION Network 4: Передача в DB "Read" значений длинн L
   RUNG wire#powerrail
      Move(in := #L1UpMMWrite, out1 => #L1UpMMRead)
      Move(in := #L1DownMMWrite, out1 => #L1DownMMRead)
   END_RUNG
   RUNG wire#powerrail
      Move(in := #L2UpMMWrite, out1 => #L2UpMMRead)
      Move(in := #L2DownMMWrite, out1 => #L2DownMMRead)
   END_RUNG
   // the same network as SCL:
   #L1UpMMRead := #L1UpMMWrite;
   #L1DownMMRead := #L1DownMMWrite;
   #L2UpMMRead := #L2UpMMWrite;
   #L2DownMMRead := #L2DownMMWrite;
END_REGION

REGION Network 5: Передача в DB "Read" установленной скорости для автоматического режима (%)
   RUNG wire#powerrail
      Move(in := #speedUpWrite, out1 => #speedUpRead)
      Move(in := #speedDownWrite, out1 => #speedDownRead)
   END_RUNG
   // the same network as SCL:
   #speedUpRead := #speedUpWrite;
   #speedDownRead := #speedDownWrite;
END_REGION

REGION Network 6: Режимы ручных переключателей преобразуются в десятичный формат
   RUNG wire#powerrail
      "binToDec"(in0 := #modeUp, in1 := #modeDown, out => #modeUpDownHMI)
   END_RUNG
   // the same network as SCL:
   "binToDec"(in0 := #modeUp, in1 := #modeDown, out => #modeUpDownHMI);
END_REGION

REGION Network 7: Положения концевиков передаются в DB "Write"
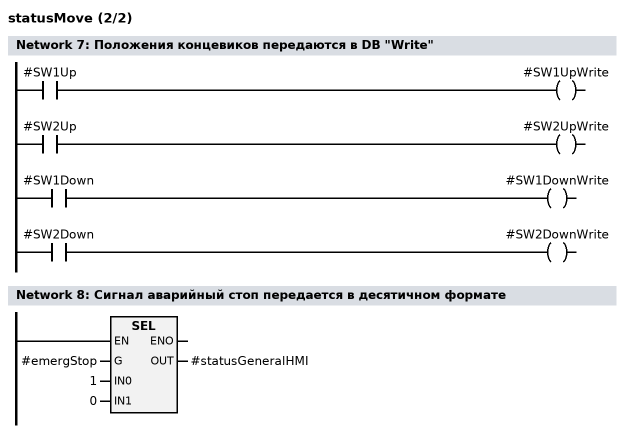
   RUNG wire#powerrail
      Contact( #SW1Up )
      Coil( #SW1UpWrite )
   END_RUNG
   RUNG wire#powerrail
      Contact( #SW2Up )
      Coil( #SW2UpWrite )
   END_RUNG
   RUNG wire#powerrail
      Contact( #SW1Down )
      Coil( #SW1DownWrite )
   END_RUNG
   RUNG wire#powerrail
      Contact( #SW2Down )
      Coil( #SW2DownWrite )
   END_RUNG
   // the same network as SCL:
   #SW1UpWrite := #SW1Up;
   #SW2UpWrite := #SW2Up;
   #SW1DownWrite := #SW1Down;
   #SW2DownWrite := #SW2Down;
END_REGION

REGION Network 8: Сигнал аварийный стоп передается в десятичном формате
   #statusGeneralHMI := SEL(G := #emergStop, IN0 := 1, IN1 := 0);
END_REGION
END_FUNCTION_BLOCK

// ===== library: MasterCopy "aprox&err" =====

FUNCTION "aprox&err" : Void   // FC1, SCL
{ S7_Optimized_Access := 'TRUE' }
VERSION : 0.1
   VAR_INPUT
      input : Int;
      in0 : Real;
      in1 : Real;
      out0 : Real;
      out1 : Real;
   END_VAR
   VAR_OUTPUT
      max : Bool;
      min : Bool;
      Out : Real;
   END_VAR
   VAR_TEMP
      input_R : Real;
   END_VAR
BEGIN
   #input_R := INT_TO_REAL(#input);
   #Out := (#input_R - #in0) * (#out1 - #out0) / (#in0 - #in0) + #out0;
   IF #Out < 0 THEN
       #min := TRUE;
       #Out := 0;
   END_IF;
   IF #Out > 100 THEN
       #max := TRUE;
       #Out := 100;
   END_IF;
END_FUNCTION

// ===== library: MasterCopy "Text_codes" =====

FUNCTION "Text_codes" : Void   // FC3, SCL
{ S7_Optimized_Access := 'TRUE' }
VERSION : 0.1
   VAR_INPUT
      initia : Bool;
      run : Bool;
      alarm : Bool;
   END_VAR
   VAR_OUTPUT
      Text_code : Int;
   END_VAR
BEGIN
   IF #initia THEN
       #Text_code := 1;
   END_IF;

   IF #run THEN
       #Text_code := 2;
   END_IF;

   IF #alarm THEN
       #Text_code := 3;
   END_IF;
END_FUNCTION

// ===== library: MasterCopy "2mux(dint)" =====

FUNCTION "2mux(dint)" : Void   // FC2, SCL
{ S7_Optimized_Access := 'TRUE' }
VERSION : 0.1
   VAR_INPUT
      adr : Bool;
      in0 : DInt;
      in1 : DInt;
   END_VAR
   VAR_OUTPUT
      out : DInt;
   END_VAR
BEGIN
   IF #adr THEN
       #out := #in1;
   ELSIF NOT #adr THEN
       #out := #in0;
   END_IF;
END_FUNCTION

// ===== library: MasterCopy "^Ch_Dint" =====

FUNCTION_BLOCK "^Ch_Dint"   // FB1, SCL
{ S7_Optimized_Access := 'TRUE' }
VERSION : 0.1
   VAR_INPUT
      in : DInt;
   END_VAR
   VAR_OUTPUT
      "^out" : Bool;
   END_VAR
   VAR
      buff : DInt;
   END_VAR
BEGIN
   IF #in <> #buff THEN
       #"^out" := true;
   ELSE
       #"^out" := false;
   END_IF;
   #buff := #in;
END_FUNCTION_BLOCK